(* IEC 61131-3 sources: pandora/pandora/aws-platform-main/aws-platform-main/configurations/base, 23 files *)

(* ---- Adaptio_IO.st ---- *)
USING Esab.Modes;

CONFIGURATION AdaptioIoMapping
    {::ifndef UNLINK_ADAPTIO_IO}
    VAR_GLOBAL
        // Adaptio
        {S7.Extern=ReadOnly}
        I_Adaptio AT %IB1000 : RawFromAdaptio;
        {S7.Extern=ReadOnly}
        Q_Adaptio AT %QB1000 : RawToAdaptio;
    END_VAR
    {::else}
    VAR_GLOBAL
        // Adaptio
        {S7.Extern=ReadWrite}
        I_Adaptio : RawFromAdaptio;
        {S7.Extern=ReadWrite}
        Q_Adaptio : RawToAdaptio;
    END_VAR
    {::endif}
END_CONFIGURATION

(* ---- B_IO.st ---- *)
USING Esab.Io;
USING Esab.WeldSystem.PowerSources;

CONFIGURATION BIoMapping
    {::ifndef UNLINK_B_IO}
    VAR_GLOBAL
        // -- B70 (Main I/O in B-cabinet) input/output starts at %X100

        // B71.1
        DI_B_System_CircuitBreaker_ServoDrives_OK AT %I100.0 : BOOL;
        DI_B_System_CircuitBreaker_ExternalConsumers_OK AT %I100.1 : BOOL;
        DI_B_System_EmergencyStop_OK AT %I100.2 : BOOL;
        DI_B_System_AirPressure_OK AT %I100.3 : BOOL;
        DI_B_RollerBed_External_Error AT %I100.4 : BOOL;
        /// Emergency stop reset button (B-cabinet)
        DI_B_PushButton_EmergencyStop_Reset AT %I100.5 : BOOL;
        // DI_SPARE AT %I100.6 : BOOL;
        // DI_SPARE AT %I100.7 : BOOL;
        DI_B_SpeedWheel_OneTurnSwitch AT %I101.0 : BOOL;
        DI_B_FluxSystem_Error AT %I101.1 : BOOL;
        DI_B_ClimateControl_Alarm AT %I101.2 : BOOL;
        // DI_SPARE AT %I101.3 : BOOL;
        // DI_SPARE AT %I101.4 : BOOL;
        // DI_SPARE AT %I101.5 : BOOL;
        // DI_SPARE AT %I101.6 : BOOL;
        // DI_SPARE AT %I101.7 : BOOL;

        // B71.2
        DI_B_PushButton_PusherRemote_WireFeed1_Down AT %I102.0 : BOOL;
        DI_B_PushButton_PusherRemote_WireFeed1_Up AT %I102.1 : BOOL;
        DI_B_PushButton_PusherRemote_WireFeed1_HighSpeed AT %I102.2 : BOOL;
        DI_B_PushButton_PusherRemote_WireFeed2_Down AT %I102.3 : BOOL;
        DI_B_PushButton_PusherRemote_WireFeed2_Up AT %I102.4 : BOOL;
        DI_B_PushButton_PusherRemote_WireFeed2_HighSpeed AT %I102.5 : BOOL;
        DI_B_PushButton_PusherRemote_WireFeed3_Down AT %I102.6 : BOOL;
        DI_B_PushButton_PusherRemote_WireFeed3_Up AT %I102.7 : BOOL;
        DI_B_PushButton_PusherRemote_WireFeed3_HighSpeed AT %I103.0 : BOOL;
        // DI_SPARE AT %I103.1 : BOOL;
        // DI_SPARE AT %I103.2 : BOOL;
        // DI_SPARE AT %I103.3 : BOOL;
        // DI_SPARE AT %I103.4 : BOOL;
        // DI_SPARE AT %I103.5 : BOOL;
        // DI_SPARE AT %I103.6 : BOOL;
        // DI_SPARE AT %I103.7 : BOOL;

        // B72.1
        DQ_B_PowerSource1_RemoteStart AT %Q100.0 : BOOL;
        DQ_B_PowerSource2_RemoteStart AT %Q100.1 : BOOL;
        DQ_B_PowerSource3_RemoteStart AT %Q100.2 : BOOL;
        DQ_B_System_RotatingWarningLight AT %Q100.3 : BOOL;
        DQ_B_FluxSystem_LowFluxWarningLight AT %Q100.4 : BOOL;
        /// This sets the reset signal to the safety relay in cabinet B.
        /// Do not use until safety investigation is complete.
        DQ_B_System_EmergencyStop_Reset AT %Q100.5 : BOOL;
        DQ_B_HighSpeed_Indicators AT %Q100.6 : BOOL;
        // DQ_SPARE AT Q100.7 : BOOL;
        // DQ_SPARE AT Q101.0 : BOOL;
        // DQ_SPARE AT Q101.1 : BOOL;
        // DQ_SPARE AT Q101.2 : BOOL;
        // DQ_SPARE AT Q101.3 : BOOL;
        // DQ_SPARE AT Q101.4 : BOOL;
        // DQ_SPARE AT Q101.5 : BOOL;
        // DQ_SPARE AT Q101.6 : BOOL;
        // DQ_SPARE AT Q101.7 : BOOL;

        // B73.1
        AI_B_EdgeSensor_Value AT %IW104 : INT;
        //AI_SPARE AT %IW106 : INT;
        //AI_SPARE AT %IW108 : INT;
        //AI_SPARE AT %IW110 : INT;

        // B74.1
        AI_B_FluxSystem_Temperature AT %IW112 : INT;
        //AI_SPARE AT %IW114 : INT;
        //AI_SPARE AT %IW116 : INT;
        //AI_SPARE AT %IW118 : INT;

        // B75.1
        AQ_B_RollerBed_SpeedReference AT %QW102 : INT;
        // AQ_SPARE AT %Q104 : INT;

        // B76.1
        DQ_B_RollerBed_Forward AT %Q106.0 : BOOL;
        DQ_B_RollerBed_Reverse AT %Q106.1 : BOOL;
        DQ_B_RollerBed_RemoteControl AT %Q106.2 : BOOL;
        // DQ_SPARE AT %Q106.3 : BOOL;

        // B77.1
        I_HighSpeedCounter AT %IB120 : RawHighSpeedCounterInputs;
        Q_HighSpeedCounter AT %QB107 : RawHighSpeedCounterOutputs;

        // B78.1
        DI_B_WireFeed1_PusherEncoder_A AT %I136.0 : BOOL;
        DI_B_WireFeed2_PusherEncoder_A AT %I136.1 : BOOL;
        DI_B_WireFeed3_PusherEncoder_A AT %I136.2 : BOOL;
        // DI_SPARE AT %I136.3 : BOOL;
        DI_B_WireFeed1_PusherEncoder_B AT %I136.4 : BOOL;
        DI_B_WireFeed2_PusherEncoder_B AT %I136.5 : BOOL;
        DI_B_WireFeed3_PusherEncoder_B AT %I136.6 : BOOL;
    END_VAR
    {::else}
    VAR_GLOBAL
        // -- B70 (Main I/O in B-cabinet) input/output starts at %X100

        // B71.1
        {S7.Extern=ReadWrite}
        DI_B_System_CircuitBreaker_ServoDrives_OK : BOOL;
        {S7.Extern=ReadWrite}
        DI_B_System_CircuitBreaker_ExternalConsumers_OK : BOOL;
        {S7.Extern=ReadWrite}
        DI_B_System_EmergencyStop_OK : BOOL;
        {S7.Extern=ReadWrite}
        DI_B_System_AirPressure_OK : BOOL;
        {S7.Extern=ReadWrite}
        DI_B_RollerBed_External_Error : BOOL;
        /// Emergency stop reset button (B-cabinet)
        {S7.Extern=ReadWrite}
        DI_B_PushButton_EmergencyStop_Reset : BOOL;
        // DI_SPARE AT %I100.6 : BOOL;
        // DI_SPARE AT %I100.7 : BOOL;
        {S7.Extern=ReadWrite}
        DI_B_SpeedWheel_OneTurnSwitch : BOOL;
        {S7.Extern=ReadWrite}
        DI_B_FluxSystem_Error : BOOL;
        {S7.Extern=ReadWrite}
        DI_B_ClimateControl_Alarm : BOOL;
        // DI_SPARE AT %I101.3 : BOOL;
        // DI_SPARE AT %I101.4 : BOOL;
        // DI_SPARE AT %I101.5 : BOOL;
        // DI_SPARE AT %I101.6 : BOOL;
        // DI_SPARE AT %I101.7 : BOOL;

        // B71.2
        {S7.Extern=ReadWrite}
        DI_B_PushButton_PusherRemote_WireFeed1_Down : BOOL;
        {S7.Extern=ReadWrite}
        DI_B_PushButton_PusherRemote_WireFeed1_Up : BOOL;
        {S7.Extern=ReadWrite}
        DI_B_PushButton_PusherRemote_WireFeed1_HighSpeed : BOOL;
        {S7.Extern=ReadWrite}
        DI_B_PushButton_PusherRemote_WireFeed2_Down : BOOL;
        {S7.Extern=ReadWrite}
        DI_B_PushButton_PusherRemote_WireFeed2_Up : BOOL;
        {S7.Extern=ReadWrite}
        DI_B_PushButton_PusherRemote_WireFeed2_HighSpeed : BOOL;
        {S7.Extern=ReadWrite}
        DI_B_PushButton_PusherRemote_WireFeed3_Down : BOOL;
        {S7.Extern=ReadWrite}
        DI_B_PushButton_PusherRemote_WireFeed3_Up : BOOL;
        {S7.Extern=ReadWrite}
        DI_B_PushButton_PusherRemote_WireFeed3_HighSpeed : BOOL;
        // DI_SPARE AT %I103.1 : BOOL;
        // DI_SPARE AT %I103.2 : BOOL;
        // DI_SPARE AT %I103.3 : BOOL;
        // DI_SPARE AT %I103.4 : BOOL;
        // DI_SPARE AT %I103.5 : BOOL;
        // DI_SPARE AT %I103.6 : BOOL;
        // DI_SPARE AT %I103.7 : BOOL;

        // B72.1
        {S7.Extern=ReadWrite}
        DQ_B_PowerSource1_RemoteStart : BOOL;
        {S7.Extern=ReadWrite}
        DQ_B_PowerSource2_RemoteStart : BOOL;
        {S7.Extern=ReadWrite}
        DQ_B_PowerSource3_RemoteStart : BOOL;
        {S7.Extern=ReadWrite}
        DQ_B_System_RotatingWarningLight : BOOL;
        {S7.Extern=ReadWrite}
        DQ_B_FluxSystem_LowFluxWarningLight : BOOL;
        /// This sets the reset signal to the safety relay in cabinet B.
        /// Do not use until safety investigation is complete.
        {S7.Extern=ReadWrite}
        DQ_B_System_EmergencyStop_Reset : BOOL;
        {S7.Extern=ReadWrite}
        DQ_B_HighSpeed_Indicators : BOOL;
        // DQ_SPARE AT Q100.7 : BOOL;
        // DQ_SPARE AT Q101.0 : BOOL;
        // DQ_SPARE AT Q101.1 : BOOL;
        // DQ_SPARE AT Q101.2 : BOOL;
        // DQ_SPARE AT Q101.3 : BOOL;
        // DQ_SPARE AT Q101.4 : BOOL;
        // DQ_SPARE AT Q101.5 : BOOL;
        // DQ_SPARE AT Q101.6 : BOOL;
        // DQ_SPARE AT Q101.7 : BOOL;

        // B73.1
        {S7.Extern=ReadWrite}
        AI_B_EdgeSensor_Value : INT;
        //AI_SPARE AT %IW106 : INT;
        //AI_SPARE AT %IW108 : INT;
        //AI_SPARE AT %IW110 : INT;

        // B74.1
        {S7.Extern=ReadWrite}
        AI_B_FluxSystem_Temperature : INT;
        //AI_SPARE AT %IW114 : INT;
        //AI_SPARE AT %IW116 : INT;
        //AI_SPARE AT %IW118 : INT;

        // B75.1
        {S7.Extern=ReadWrite}
        AQ_B_RollerBed_SpeedReference : INT;
        // AQ_SPARE AT %Q104 : INT;

        // B76.1
        {S7.Extern=ReadWrite}
        DQ_B_RollerBed_Forward : BOOL;
        {S7.Extern=ReadWrite}
        DQ_B_RollerBed_Reverse : BOOL;
        {S7.Extern=ReadWrite}
        DQ_B_RollerBed_RemoteControl : BOOL;
        // DQ_SPARE AT %Q106.3 : BOOL;

        // B77.1
        {S7.Extern=ReadWrite}
        I_HighSpeedCounter AT %MB100 : RawHighSpeedCounterInputs;
        {S7.Extern=ReadWrite}
        Q_HighSpeedCounter AT %MB150: RawHighSpeedCounterOutputs;

        // B78.1
        {S7.Extern=ReadWrite}
        DI_B_WireFeed1_PusherEncoder_A : BOOL;
        {S7.Extern=ReadWrite}
        DI_B_WireFeed2_PusherEncoder_A : BOOL;
        {S7.Extern=ReadWrite}
        DI_B_WireFeed3_PusherEncoder_A : BOOL;
        // DI_SPARE AT %I136.3 : BOOL;
        {S7.Extern=ReadWrite}
        DI_B_WireFeed1_PusherEncoder_B : BOOL;
        {S7.Extern=ReadWrite}
        DI_B_WireFeed2_PusherEncoder_B : BOOL;
        {S7.Extern=ReadWrite}
        DI_B_WireFeed3_PusherEncoder_B : BOOL;
    END_VAR
    {::endif}

END_CONFIGURATION

(* ---- C_IO.st ---- *)
CONFIGURATION CIoMapping
    {::ifndef UNLINK_C_IO}
    VAR_GLOBAL
        // -- C1 (Button box located at welding head) input/output starts at %X50
        // NOTE: The actual buttons are in the reverse order compared to I/O-addressing

        // C2
        /// Emergency stop reset button (C-cabinet)
        DI_C_PushButton_EmergencyStop_Reset AT %I59.0 : BOOL;
        /// Emergency stop reset button LED (C-cabinet)
        DQ_C_PushButton_EmergencyStop_Reset AT %Q59.0 : BOOL;

        // C3
        DI_C_PushButton_FluxSystem_Release AT %I58.0 : BOOL;
        DQ_C_PushButton_FluxSystem_Release AT %Q58.0 : BOOL;

        // C4
        DI_C_PushButton_HighSpeed AT %I57.0 : BOOL;
        DQ_C_PushButton_HighSpeed AT %Q57.0 : BOOL;

        // C5
        DI_C_PushButton_WireFeed1_Up AT %I56.0 : BOOL;
        DI_C_PushButton_WireFeed1_Down AT %I56.1 : BOOL;

        // C6
        DI_C_PushButton_WireFeed2_Up AT %I55.0 : BOOL;
        DI_C_PushButton_WireFeed2_Down AT %I55.1 : BOOL;

        // C7
        DI_C_PushButton_WireFeed3_Up AT %I54.0 : BOOL;
        DI_C_PushButton_WireFeed3_Down AT %I54.1 : BOOL;

        // C8 (Joystick) + C9 (Wired to the command module)
        DI_C_PushButton_TrackingOff AT %I50.0 : BOOL;
        DQ_C_PushButton_TrackingOff AT %Q50.0 : BOOL;
        DI_C_MotionJoystick_Up AT %I50.2 : BOOL;
        DI_C_MotionJoystick_Down AT %I50.3 : BOOL;
        DI_C_MotionJoystick_Triangle AT %I50.4 : BOOL;
        DI_C_MotionJoystick_Square AT %I50.5 : BOOL;

        // C10
        DI_C_PushButton_Tilt_Left AT %I53.0 : BOOL;
        DI_C_PushButton_Tilt_Right AT %I53.1 : BOOL;
    END_VAR
    {::else}
    VAR_GLOBAL
        // -- C1 (Button box located at welding head) input/output starts at %X50
        // NOTE: The actual buttons are in the reverse order compared to I/O-addressing

        // C2
        /// Emergency stop reset button (C-cabinet)
        {S7.Extern=ReadWrite}
        DI_C_PushButton_EmergencyStop_Reset : BOOL;
        /// Emergency stop reset button LED (C-cabinet)
        {S7.Extern=ReadWrite}
        DQ_C_PushButton_EmergencyStop_Reset : BOOL;

        // C3
        {S7.Extern=ReadWrite}
        DI_C_PushButton_FluxSystem_Release : BOOL;
        {S7.Extern=ReadWrite}
        DQ_C_PushButton_FluxSystem_Release : BOOL;

        // C4
        {S7.Extern=ReadWrite}
        DI_C_PushButton_HighSpeed : BOOL;
        {S7.Extern=ReadWrite}
        DQ_C_PushButton_HighSpeed : BOOL;

        // C5
        {S7.Extern=ReadWrite}
        DI_C_PushButton_WireFeed1_Up : BOOL;
        {S7.Extern=ReadWrite}
        DI_C_PushButton_WireFeed1_Down : BOOL;

        // C6
        {S7.Extern=ReadWrite}
        DI_C_PushButton_WireFeed2_Up : BOOL;
        {S7.Extern=ReadWrite}
        DI_C_PushButton_WireFeed2_Down : BOOL;

        // C7
        {S7.Extern=ReadWrite}
        DI_C_PushButton_WireFeed3_Up : BOOL;
        {S7.Extern=ReadWrite}
        DI_C_PushButton_WireFeed3_Down : BOOL;

        // C8 (Joystick) + C9 (Wired to the command module)
        {S7.Extern=ReadWrite}
        DI_C_PushButton_TrackingOff : BOOL;
        {S7.Extern=ReadWrite}
        DQ_C_PushButton_TrackingOff : BOOL;
        {S7.Extern=ReadWrite}
        DI_C_MotionJoystick_Up : BOOL;
        {S7.Extern=ReadWrite}
        DI_C_MotionJoystick_Down : BOOL;
        {S7.Extern=ReadWrite}
        DI_C_MotionJoystick_Triangle : BOOL;
        {S7.Extern=ReadWrite}
        DI_C_MotionJoystick_Square : BOOL;

        // C10
        {S7.Extern=ReadWrite}
        DI_C_PushButton_Tilt_Left : BOOL;
        {S7.Extern=ReadWrite}
        DI_C_PushButton_Tilt_Right : BOOL;
    END_VAR
    {::endif}
END_CONFIGURATION

(* ---- GlobalState.st ---- *)
USING Esab.WeldSystem.Flux;
USING Esab.Utils.Alarming;
USING Esab.Utils.Assets;
USING Esab.Modes;

USING Siemens.Simatic.S71500.Tasks;
USING Siemens.Simatic.S71500.Alarming;

CONFIGURATION GlobalStateConfiguration

    // Constants
    VAR_GLOBAL CONSTANT
    END_VAR

    // Objects
    VAR_GLOBAL
        {S7.Extern=Read}
        GlobalState : Esab.GlobalState;
    END_VAR

    // Alarms
    VAR_GLOBAL
        GlobalStateSetupAlarmWrapper : AlarmWrapper;
        {S7.Alarm = NoAck, "Global state: Setup error."}
        GlobalStateSetupAlarm : ProgramAlarm;
    END_VAR

    // Interface
    VAR_GLOBAL
    END_VAR
END_CONFIGURATION

FUNCTION InitializeGlobalState
    VAR_INPUT
        assetsManager : IAssetsManager;
    END_VAR

    VAR_EXTERNAL
        GlobalState : Esab.GlobalState;

        GlobalStateSetupAlarmWrapper : AlarmWrapper;
        GlobalStateSetupAlarm : ProgramAlarm;
    END_VAR

    GlobalStateSetupAlarmWrapper.Setup(REF(GlobalStateSetupAlarm));

    GlobalState.Setup(assetsManager, GlobalStateSetupAlarmWrapper);

    GlobalState.SetIdentifier(Esab.AssetIdentifier#GlobalState);
    assetsManager.RegisterAsset(REF(GlobalState));

    // By default we set the GlobalState mode to be Adaptio
    GlobalState.SetMode(Esab.AwsPlatformMode#Adaptio);
END_FUNCTION

(* ---- H_IO.st ---- *)
CONFIGURATION HIoMapping
    {::ifndef UNLINK_H_IO}
    VAR_GLOBAL
        // -- H1 (Weld head I/O) input/output starts at %X60

        // H2.1
        DI_H_SlideCrossHorizontal_LimitSwitch_Triangle AT %I60.0 : BOOL;
        DI_H_SlideCrossHorizontal_LimitSwitch_Square AT %I60.1 : BOOL;
        DI_H_SlideCrossVertical_LimitSwitch_Up AT %I60.2 : BOOL;
        DI_H_SlideCrossVertical_LimitSwitch_Down AT %I60.3 : BOOL;
        DI_H_Tilt_LimitSwitch_Left AT %I60.4 : BOOL;
        DI_H_Tilt_LimitSwitch_Right AT %I60.5 : BOOL;
        // DI_SPARE AT %I60.6 : BOOL;
        // DI_SPARE AT %I60.7 : BOOL;

        // H3.1
        AI_H_Pyrometer_Value AT %IW61 : INT;
        AI_H_HeightSensor_Value AT %IW63 : INT;
        // AI_SPARE AT %IW65 : INT;
        // AI_SPARE AT %IW67 : INT;

        // H4.1
        DQ_H_LaserPointer_Enable AT %Q69.0 : BOOL;
        DQ_H_System_Water_WarningLight AT %Q69.1 : BOOL;
        // DQ_SPARE AT %!69.2 : BOOL;
        // DQ_SPARE AT %!69.3 : BOOL;
        // DQ_SPARE AT %!69.4 : BOOL;
        // DQ_SPARE AT %!69.5 : BOOL;
        DQ_H_Scanner_LaserLine_Enable AT %Q69.6 : BOOL;
        DQ_H_Scanner_Camera_Enable AT %Q69.7 : BOOL;

        // H4.2
        DQ_H_FluxSystem_Recover AT %Q70.0 : BOOL;
        DQ_H_FluxSystem_Release AT %Q70.1 : BOOL;
        DQ_H_Scanner_AirFlow_Enable AT %Q70.2 : BOOL;
        DQ_H_FluxSystem_NozzleRotation AT %Q70.3 : BOOL;
        // DQ_SPARE AT %Q70.4 : BOOL;
        // DQ_SPARE AT %Q70.5 : BOOL;
        // DQ_SPARE AT %Q70.6 : BOOL;
        // DQ_SPARE AT %Q70.7 : BOOL;

        // H5.1
        DQ_H_Camera_Lamp1_Enable AT %Q71.0 : BOOL;
        DQ_H_Camera_Lamp2_Enable AT %Q71.1 : BOOL;
        DQ_H_FloodLight1_Enable AT %Q71.2 : BOOL;
        DQ_H_FloodLight2_Enable AT %Q71.3 : BOOL;
    END_VAR
    {::else}
    VAR_GLOBAL
        // -- H1 (Weld head I/O) input/output starts at %X60

        // H2.1
        {S7.Extern=ReadWrite}
        DI_H_SlideCrossHorizontal_LimitSwitch_Triangle : BOOL;
        {S7.Extern=ReadWrite}
        DI_H_SlideCrossHorizontal_LimitSwitch_Square : BOOL;
        {S7.Extern=ReadWrite}
        DI_H_SlideCrossVertical_LimitSwitch_Up : BOOL;
        {S7.Extern=ReadWrite}
        DI_H_SlideCrossVertical_LimitSwitch_Down : BOOL;
        {S7.Extern=ReadWrite}
        DI_H_Tilt_LimitSwitch_Left : BOOL;
        {S7.Extern=ReadWrite}
        DI_H_Tilt_LimitSwitch_Right : BOOL;
        // DI_SPARE AT %I60.6 : BOOL;
        // DI_SPARE AT %I60.7 : BOOL;

        // H3.1
        {S7.Extern=ReadWrite}
        AI_H_Pyrometer_Value : INT;
        {S7.Extern=ReadWrite}
        AI_H_HeightSensor_Value : INT;
        // AI_SPARE AT %IW65 : INT;
        // AI_SPARE AT %IW67 : INT;

        // H4.1
        {S7.Extern=ReadWrite}
        DQ_H_LaserPointer_Enable : BOOL;
        {S7.Extern=ReadWrite}
        DQ_H_System_Water_WarningLight : BOOL;
        // DQ_SPARE AT %!69.2 : BOOL;
        // DQ_SPARE AT %!69.3 : BOOL;
        // DQ_SPARE AT %!69.4 : BOOL;
        // DQ_SPARE AT %!69.5 : BOOL;
        {S7.Extern=ReadWrite}
        DQ_H_Scanner_LaserLine_Enable : BOOL;
        {S7.Extern=ReadWrite}
        DQ_H_Scanner_Camera_Enable : BOOL;

        // H4.2
        {S7.Extern=ReadWrite}
        DQ_H_FluxSystem_Recover : BOOL;
        {S7.Extern=ReadWrite}
        DQ_H_FluxSystem_Release : BOOL;
        {S7.Extern=ReadWrite}
        DQ_H_Scanner_AirFlow_Enable : BOOL;
        {S7.Extern=ReadWrite}
        DQ_H_FluxSystem_NozzleRotation : BOOL;
        // DQ_SPARE AT %Q70.4 : BOOL;
        // DQ_SPARE AT %Q70.5 : BOOL;
        // DQ_SPARE AT %Q70.6 : BOOL;
        // DQ_SPARE AT %Q70.7 : BOOL;

        // H5.1
        {S7.Extern=ReadWrite}
        DQ_H_Camera_Lamp1_Enable : BOOL;
        {S7.Extern=ReadWrite}
        DQ_H_Camera_Lamp2_Enable : BOOL;
        {S7.Extern=ReadWrite}
        DQ_H_FloodLight1_Enable : BOOL;
        {S7.Extern=ReadWrite}
        DQ_H_FloodLight2_Enable : BOOL;
    END_VAR
    {::endif}
END_CONFIGURATION

(* ---- P_IO.st ---- *)
CONFIGURATION IoMapping
    {::ifndef UNLINK_P_IO}
    VAR_GLOBAL
        // -- P1 (Button box below the main HMI screen) input/output starts at %X30
        // NOTE: The actual buttons are in the reverse order compared to I/O-addressing

        // P2 (Emergency stop reset)
        DI_P_PushButton_EmergencyStop_Reset AT %I42.0 : BOOL;
        DQ_P_PushButton_EmergencyStop_Reset AT %Q42.0 : BOOL;

        // P3 (Flux release/down)
        DI_P_PushButton_FluxSystem_Release AT %I41.0 : BOOL;
        DQ_P_PushButton_FluxSystem_Release AT %Q41.0 : BOOL;

        // P4 (Flux recover/suction)
        DI_P_PushButton_FluxSystem_Recover AT %I40.0 : BOOL;
        DQ_P_PushButton_FluxSystem_Recover AT %Q40.0 : BOOL;

        // P5 (High speed selection)
        DI_P_PushButton_HighSpeed AT %I39.0 : BOOL;
        DQ_P_PushButton_HighSpeed AT %Q39.0 : BOOL;

        // P6 (Wire feed 1 + 3)
        /// NOTE: This also controls WF 3 Up through mode select
        DI_P_PushButton_WireFeed1_Up AT %I38.0 : BOOL;
        /// NOTE: This also controls WF 3 Down through mode select
        DI_P_PushButton_WireFeed1_Down AT %I38.1 : BOOL;

        // P7
        DI_P_PushButton_WireFeed2_Up AT %I37.0 : BOOL;
        DI_P_PushButton_WireFeed2_Down AT %I37.1 : BOOL;

        // P8 (Joystick) + P9 (Axis selection)
        DI_P_MotionJoystick_AxisSelection AT %I30.0 : BOOL;
        DQ_P_MotionJoystick_AxisSelection AT %Q30.0 : BOOL;
        DI_P_MotionJoystick_Up AT %I30.2 : BOOL;
        DI_P_MotionJoystick_Down AT %I30.3 : BOOL;
        DI_P_MotionJoystick_Triangle AT %I30.4 : BOOL;
        DI_P_MotionJoystick_Square AT %I30.5 : BOOL;

        // P10 (Axis selection triangle/square)
        DI_P_PushButton_AxisJog_AxisSelection AT %I36.0 : BOOL;
        DQ_P_PushButton_AxisJog_AxisSelection AT %Q36.0 : BOOL;

        // P11 (Axis triangle/square)
        DI_P_PushButton_AxisJog_Triangle AT %I35.0 : BOOL;
        DI_P_PushButton_AxisJog_Square AT %I35.1 : BOOL;

        // P12 (Start)
        DI_P_PushButton_Start AT %I34.0 : BOOL;
        DQ_P_PushButton_Start AT %Q34.0 : BOOL;

        // P13 (Stop)
        DI_P_PushButton_Stop AT %I33.0 : BOOL;
        DQ_P_PushButton_Stop AT %Q33.0 : BOOL;
    END_VAR
    {::else}
    VAR_GLOBAL
        // -- P1 (Button box below the main HMI screen) input/output starts at %X30
        // NOTE: The actual buttons are in the reverse order compared to I/O-addressing

        // P2 (Emergency stop reset)
        {S7.Extern=ReadWrite}
        DI_P_PushButton_EmergencyStop_Reset : BOOL;
        {S7.Extern=ReadWrite}
        DQ_P_PushButton_EmergencyStop_Reset : BOOL;

        // P3 (Flux release/down)
        {S7.Extern=ReadWrite}
        DI_P_PushButton_FluxSystem_Release : BOOL;
        {S7.Extern=ReadWrite}
        DQ_P_PushButton_FluxSystem_Release : BOOL;

        // P4 (Flux recover/suction)
        {S7.Extern=ReadWrite}
        DI_P_PushButton_FluxSystem_Recover : BOOL;
        {S7.Extern=ReadWrite}
        DQ_P_PushButton_FluxSystem_Recover : BOOL;

        // P5 (High speed selection)
        {S7.Extern=ReadWrite}
        DI_P_PushButton_HighSpeed : BOOL;
        {S7.Extern=ReadWrite}
        DQ_P_PushButton_HighSpeed : BOOL;

        // P6 (Wire feed 1 + 3)
        /// NOTE: This also controls WF 3 Up through mode select
        {S7.Extern=ReadWrite}
        DI_P_PushButton_WireFeed1_Up : BOOL;
        /// NOTE: This also controls WF 3 Down through mode select
        {S7.Extern=ReadWrite}
        DI_P_PushButton_WireFeed1_Down : BOOL;

        // P7
        {S7.Extern=ReadWrite}
        DI_P_PushButton_WireFeed2_Up : BOOL;
        {S7.Extern=ReadWrite}
        DI_P_PushButton_WireFeed2_Down : BOOL;

        // P8 (Joystick) + P9 (Axis selection)
        {S7.Extern=ReadWrite}
        DI_P_MotionJoystick_AxisSelection : BOOL;
        {S7.Extern=ReadWrite}
        DQ_P_MotionJoystick_AxisSelection : BOOL;
        {S7.Extern=ReadWrite}
        DI_P_MotionJoystick_Up : BOOL;
        {S7.Extern=ReadWrite}
        DI_P_MotionJoystick_Down : BOOL;
        {S7.Extern=ReadWrite}
        DI_P_MotionJoystick_Triangle : BOOL;
        {S7.Extern=ReadWrite}
        DI_P_MotionJoystick_Square : BOOL;

        // P10 (Axis selection triangle/square)
        {S7.Extern=ReadWrite}
        DI_P_PushButton_AxisJog_AxisSelection : BOOL;
        {S7.Extern=ReadWrite}
        DQ_P_PushButton_AxisJog_AxisSelection : BOOL;

        // P11 (Axis triangle/square)
        {S7.Extern=ReadWrite}
        DI_P_PushButton_AxisJog_Triangle : BOOL;
        {S7.Extern=ReadWrite}
        DI_P_PushButton_AxisJog_Square : BOOL;

        // P12 (Start)
        {S7.Extern=ReadWrite}
        DI_P_PushButton_Start : BOOL;
        {S7.Extern=ReadWrite}
        DQ_P_PushButton_Start : BOOL;

        // P13 (Stop)
        {S7.Extern=ReadWrite}
        DI_P_PushButton_Stop : BOOL;
        {S7.Extern=ReadWrite}
        DQ_P_PushButton_Stop : BOOL;
    END_VAR
    {::endif}
END_CONFIGURATION

(* ---- PowerSources_IO.st ---- *)
USING Esab.WeldSystem.PowerSources;

CONFIGURATION PowerSourcesIoMapping
    {::ifndef UNLINK_POWERSOURCES_IO}
    VAR_GLOBAL
        // Power sources
        I_Pab1 AT %IB500 : RawPabToController;
        Q_Pab1 AT %QB500 : RawControllerToPab;
        I_Pab2 AT %IB600 : RawPabToController;
        Q_Pab2 AT %QB600 : RawControllerToPab;
    END_VAR
    {::else}
    VAR_GLOBAL
        // Power sources
        {S7.Extern=ReadWrite}
        I_Pab1 : RawPabToController;
        {S7.Extern=ReadWrite}
        Q_Pab1 : RawControllerToPab;
        {S7.Extern=ReadWrite}
        I_Pab2 : RawPabToController;
        {S7.Extern=ReadWrite}
        Q_Pab2 : RawControllerToPab;
    END_VAR
    {::endif}
END_CONFIGURATION

(* ---- SlideCrossAxis.st ---- *)
USING Esab.Motion;
USING Esab.Utils.Assets;

CONFIGURATION SlideCrossConfiguration
    // Constants
    VAR_GLOBAL CONSTANT
        HORIZONTAL_SLIDE_AXIS_DB : Siemens.Simatic.S71500.MotionControl.Native.DB_ANY := UINT#1;
        VERTICAL_SLIDE_AXIS_DB : Siemens.Simatic.S71500.MotionControl.Native.DB_ANY := UINT#2;
    END_VAR

    // Objects
    VAR_GLOBAL
        Technology : TechnologyObjects;
        HorizontalSlideAxis : ToPosAxis;
        HorizontalSlideAxisRuntimeParameters : AxisRuntimeParameters;
        VerticalSlideAxis : ToPosAxis;
        VerticalSlideAxisRuntimeParameters : AxisRuntimeParameters;
    END_VAR

    // Alarms
    VAR_GLOBAL
    END_VAR

    // Interface
    VAR_GLOBAL
    END_VAR
END_CONFIGURATION

FUNCTION InitializeSlideCrossAxis
    VAR_INPUT
        assetsManager : IAssetsManager;
    END_VAR

    VAR_EXTERNAL CONSTANT
        HORIZONTAL_SLIDE_AXIS_DB : Siemens.Simatic.S71500.MotionControl.Native.DB_ANY;
        VERTICAL_SLIDE_AXIS_DB : Siemens.Simatic.S71500.MotionControl.Native.DB_ANY;
    END_VAR

    VAR_EXTERNAL
        Technology : TechnologyObjects;
        HorizontalSlideAxis : ToPosAxis;
        HorizontalSlideAxisRuntimeParameters : AxisRuntimeParameters;
        VerticalSlideAxis : ToPosAxis;
        VerticalSlideAxisRuntimeParameters : AxisRuntimeParameters;
    END_VAR

    Technology.Setup(HORIZONTAL_SLIDE_AXIS_DB, VERTICAL_SLIDE_AXIS_DB);

    IF Technology.IsAttached() THEN
        HorizontalSlideAxis.Setup(Technology.GetHorizontalSlideAxis(), REF(HorizontalSlideAxisRuntimeParameters));
        VerticalSlideAxis.Setup(Technology.GetVerticalSlideAxis(), REF(VerticalSlideAxisRuntimeParameters));

        HorizontalSlideAxis.SetIdentifier(Esab.AssetIdentifier#HorizontalSlideAxis);
        VerticalSlideAxis.SetIdentifier(Esab.AssetIdentifier#VerticalSlideAxis);
        assetsManager.RegisterAsset(REF(HorizontalSlideAxis));
        assetsManager.RegisterAsset(REF(VerticalSlideAxis));
    END_IF;
END_FUNCTION

(* ---- Ups1600_IO.st ---- *)
USING Esab.Utils.Power;

CONFIGURATION Ups1600IoMapping

    {::ifndef UNLINK_UPS_IO}
    VAR_GLOBAL
        {S7.Extern=ReadOnly}
        I_Ups AT %IB0 : RawFromUps1600;
    END_VAR
    {::else}
    VAR_GLOBAL
        {S7.Extern=ReadWrite}
        I_Ups : RawFromUps1600;
    END_VAR
    {::endif}

END_CONFIGURATION

(* ---- WeldHeadManipulator.st ---- *)
USING Esab.Utils.Alarming;
USING Esab.Utils.Assets;
USING Esab.Motion;

USING Siemens.Simatic.S71500.Tasks;
USING Siemens.Simatic.S71500.Alarming;

CONFIGURATION WeldHeadManipulatorConfiguration

    // Constants
    VAR_GLOBAL CONSTANT
    END_VAR

    // Objects
    VAR_GLOBAL
        {S7.Extern=Read}
        WeldHeadManipulator : WeldHeadManipulator;
    END_VAR

    // Alarms
    VAR_GLOBAL
        WeldHeadManipulatorSetupAlarmWrapper : AlarmWrapper;
        {S7.Alarm = NoAck, "Global state: Setup error."}
        WeldHeadManipulatorSetupAlarm : ProgramAlarm;
    END_VAR

    // Interface
    VAR_GLOBAL
    END_VAR

    VAR_GLOBAL RETAIN
        WeldHeadManipulatorRuntimeParameters : WeldHeadManipulatorRuntimeParameters;
        WeldHeadManipulatorHardwareConfiguration : WeldHeadManipulatorHardwareConfiguration;
    END_VAR
END_CONFIGURATION

FUNCTION InitializeWeldHeadManipulator
    VAR_INPUT
        assetsManager : IAssetsManager;
    END_VAR

    VAR_EXTERNAL
        WeldHeadManipulator : WeldHeadManipulator;
        WeldHeadManipulatorRuntimeParameters : WeldHeadManipulatorRuntimeParameters;
        WeldHeadManipulatorHardwareConfiguration : WeldHeadManipulatorHardwareConfiguration;

        WeldHeadManipulatorSetupAlarmWrapper : AlarmWrapper;
        WeldHeadManipulatorSetupAlarm : ProgramAlarm;
    END_VAR

    WeldHeadManipulatorSetupAlarmWrapper.Setup(REF(WeldHeadManipulatorSetupAlarm));

    WeldHeadManipulator.Setup(REF(WeldHeadManipulatorRuntimeParameters),
                              REF(WeldHeadManipulatorHardwareConfiguration),
                              assetsManager,
                              WeldHeadManipulatorSetupAlarmWrapper);

    WeldHeadManipulator.SetIdentifier(Esab.AssetIdentifier#WeldHeadManipulator);
    assetsManager.RegisterAsset(REF(WeldHeadManipulator));
END_FUNCTION

(* ---- WeldSystemOrchestrator.st ---- *)
USING Esab.Utils.Alarming;
USING Esab.Utils.Assets;
USING Esab.WeldSystem;

USING Siemens.Simatic.S71500.Alarming;

CONFIGURATION WeldSystemOrchestratorConfiguration

    // Constants
    VAR_GLOBAL CONSTANT
    END_VAR

    // Objects
    VAR_GLOBAL
        WeldSystemOrchestrator : WeldSystemOrchestrator;
    END_VAR

    // Alarms
    VAR_GLOBAL
        WeldSystemOrchestratorSetupAlarmWrapper : AlarmWrapper;
        {S7.Alarm = NoAck, "Weld system: Setup error."}
        WeldSystemOrchestratorSetupAlarm : ProgramAlarm;
    END_VAR

    // Interface
    VAR_GLOBAL
    END_VAR

    VAR_GLOBAL RETAIN
        WeldSystemOrchestratorRuntimeParameters : WeldSystemOrchestratorRuntimeParameters;
        WeldSystemOrchestratorHardwareConfiguration : WeldSystemOrchestratorHardwareConfiguration;
    END_VAR
END_CONFIGURATION

FUNCTION InitializeMultiWeldSystem
    VAR_INPUT
        assetsManager : IAssetsManager;
    END_VAR

    VAR_EXTERNAL
        WeldSystemOrchestrator : WeldSystemOrchestrator;
        WeldSystemOrchestratorRuntimeParameters : WeldSystemOrchestratorRuntimeParameters;
        WeldSystemOrchestratorHardwareConfiguration : WeldSystemOrchestratorHardwareConfiguration;
        WeldSystemOrchestratorSetupAlarmWrapper : AlarmWrapper;
        WeldSystemOrchestratorSetupAlarm : ProgramAlarm;
    END_VAR

    WeldSystemOrchestratorSetupAlarmWrapper.Setup(REF(WeldSystemOrchestratorSetupAlarm));

    WeldSystemOrchestrator.Setup(REF(WeldSystemOrchestratorRuntimeParameters),
                                 REF(WeldSystemOrchestratorHardwareConfiguration),
                                 assetsManager,
                                 WeldSystemOrchestratorSetupAlarmWrapper);

    WeldSystemOrchestrator.SetIdentifier(Esab.AssetIdentifier#WeldSystemOrchestrator);
    assetsManager.RegisterAsset(REF(WeldSystemOrchestrator));
END_FUNCTION

(* ---- Adaptio.st ---- *)
USING Esab.Modes;
USING Esab.Utils.Alarming;
USING Esab.Utils.Assets;
USING Esab.Utils.Heartbeat;
USING Esab.Utils.Timer;

USING Siemens.Simatic.S71500.Tasks;
USING Siemens.Simatic.S71500.Alarming;

CONFIGURATION AdaptioSystemConfiguration

    TASK AdaptioIoTask : ProgramCycle;

    PROGRAM AdaptioIoReadWrite WITH AdaptioIoTask: AdaptioIoReadWrite;

    // Constants
    VAR_GLOBAL CONSTANT
    END_VAR

    // Objects
    VAR_GLOBAL
        {S7.Extern=Read}
        Adaptio : Adaptio;
        AdaptioRuntimeParameters : AdaptioRuntimeParameters;
        AdaptioWeldSequence : AdaptioWeldSequence;
        AdaptioWeldSequenceStateTimer : ITimer;
        AdaptioHeartbeat : IncrementingHeartbeat;
        AdaptioRequestTimer : OnDelay;
        AdaptioJoystickClickTimer : OnDelay;
        AdaptioWeldingStateTimer : OnDelay;
        AdaptioHeartbeatTimer : OnDelay;
    END_VAR

    // Alarms
    VAR_GLOBAL
        AdaptioHeartbeatAlarmWrapper : AlarmWrapper;
        {S7.Alarm = NoAck, "Adaptio: Heartbeat missing."}
        AdaptioHeartbeatAlarm : ProgramAlarm;

        AdaptioSetupAlarmWrapper : AlarmWrapper;
        {S7.Alarm = NoAck, "Adaptio: Setup error."}
        AdaptioSetupAlarm : ProgramAlarm;
    END_VAR

    // Interface
    VAR_GLOBAL
        {S7.Extern=ReadWrite}
        AdaptioIo : AdaptioIo;
    END_VAR
END_CONFIGURATION

FUNCTION InitializeAdaptio
    VAR_INPUT
        assetsManager : IAssetsManager;
    END_VAR

    VAR_EXTERNAL
        AdaptioIo : AdaptioIo;

        Adaptio : Adaptio;
        AdaptioRuntimeParameters : AdaptioRuntimeParameters;
        AdaptioWeldSequence : AdaptioWeldSequence;
        AdaptioWeldSequenceStateTimer : ITimer;
        AdaptioHeartbeat : IncrementingHeartbeat;
        AdaptioRequestTimer : OnDelay;
        AdaptioJoystickClickTimer : OnDelay;
        AdaptioWeldingStateTimer : OnDelay;
        AdaptioHeartbeatTimer : OnDelay;

        AdaptioHeartbeatAlarmWrapper : AlarmWrapper;
        AdaptioHeartbeatAlarm : ProgramAlarm;

        AdaptioSetupAlarmWrapper : AlarmWrapper;
        AdaptioSetupAlarm : ProgramAlarm;
    END_VAR

    AdaptioWeldSequence.Setup(AdaptioWeldSequenceStateTimer); // Weld axis and orchestrator is set inside the Adaptio manager
    AdaptioHeartbeatAlarmWrapper.Setup(REF(AdaptioHeartbeatAlarm));
    AdaptioSetupAlarmWrapper.Setup(REF(AdaptioSetupAlarm));

    AdaptioHeartbeat.Setup(AdaptioIo.FromAdaptio.SystemControl.Heartbeat,
                           AdaptioIo.ToAdaptio.SystemControl.Heartbeat,
                           AdaptioHeartbeatTimer,
                           AdaptioHeartbeatAlarmWrapper);

    Adaptio.Setup(REF(AdaptioIo),
                  REF(AdaptioRuntimeParameters),
                  assetsManager,
                  AdaptioWeldSequence,
                  AdaptioHeartbeat,
                  AdaptioRequestTimer,
                  AdaptioJoystickClickTimer,
                  AdaptioSetupAlarmWrapper);
END_FUNCTION

PROGRAM AdaptioIoReadWrite
    VAR_EXTERNAL
        AdaptioIo : AdaptioIo;
        I_Adaptio : RawFromAdaptio;
        Q_Adaptio : RawToAdaptio;
    END_VAR

    AdaptioIo.FromAdaptio.SystemControl.Heartbeat.Read(I_Adaptio.SystemControl.Heartbeat);

    AdaptioIo.FromAdaptio.WeldControl.Start.Read(I_Adaptio.WeldControl.Start);
    AdaptioIo.FromAdaptio.WeldControl.Stop.Read(I_Adaptio.WeldControl.Stop);
    AdaptioIo.FromAdaptio.WeldControl.QuickStop.Read(I_Adaptio.WeldControl.QuickStop);

    AdaptioIo.FromAdaptio.PowerSource1.Enable.Read(I_Adaptio.PowerSource1.Enable);
    AdaptioIo.FromAdaptio.PowerSource1.ActiveAreaSelect.Read(I_Adaptio.PowerSource1.ActiveAreaSelect);
    AdaptioIo.FromAdaptio.PowerSource1.SwitchAreas.Read(I_Adaptio.PowerSource1.SwitchAreas);
    AdaptioIo.FromAdaptio.PowerSource1.Voltage.Read(I_Adaptio.PowerSource1.Voltage);
    AdaptioIo.FromAdaptio.PowerSource1.Current.Read(I_Adaptio.PowerSource1.Current);
    AdaptioIo.FromAdaptio.PowerSource1.WireSpeed.Read(I_Adaptio.PowerSource1.WireSpeed);
    AdaptioIo.FromAdaptio.PowerSource1.RegulationType.Read(I_Adaptio.PowerSource1.RegulationType);
    AdaptioIo.FromAdaptio.PowerSource1.WeldMethod.Read(I_Adaptio.PowerSource1.WeldMethod);
    AdaptioIo.FromAdaptio.PowerSource1.AcFrequency.Read(I_Adaptio.PowerSource1.AcFrequency);
    AdaptioIo.FromAdaptio.PowerSource1.AcBalance.Read(I_Adaptio.PowerSource1.AcBalance);
    AdaptioIo.FromAdaptio.PowerSource1.AcOffset.Read(I_Adaptio.PowerSource1.AcOffset);
    AdaptioIo.FromAdaptio.PowerSource1.AcPhaseShift.Read(I_Adaptio.PowerSource1.AcPhaseShift);
    AdaptioIo.FromAdaptio.PowerSource1.StartAdjust.Read(I_Adaptio.PowerSource1.StartAdjust);
    AdaptioIo.FromAdaptio.PowerSource1.RegulationDynamics.Read(I_Adaptio.PowerSource1.RegulationDynamics);
    AdaptioIo.FromAdaptio.PowerSource1.RegulationInductance.Read(I_Adaptio.PowerSource1.RegulationInductance);
    AdaptioIo.FromAdaptio.PowerSource1.IceWireSpeed.Read(I_Adaptio.PowerSource1.IceWireSpeed);

    AdaptioIo.FromAdaptio.PowerSource2.Enable.Read(I_Adaptio.PowerSource2.Enable);
    AdaptioIo.FromAdaptio.PowerSource2.ActiveAreaSelect.Read(I_Adaptio.PowerSource2.ActiveAreaSelect);
    AdaptioIo.FromAdaptio.PowerSource2.SwitchAreas.Read(I_Adaptio.PowerSource2.SwitchAreas);
    AdaptioIo.FromAdaptio.PowerSource2.Voltage.Read(I_Adaptio.PowerSource2.Voltage);
    AdaptioIo.FromAdaptio.PowerSource2.Current.Read(I_Adaptio.PowerSource2.Current);
    AdaptioIo.FromAdaptio.PowerSource2.WireSpeed.Read(I_Adaptio.PowerSource2.WireSpeed);
    AdaptioIo.FromAdaptio.PowerSource2.RegulationType.Read(I_Adaptio.PowerSource2.RegulationType);
    AdaptioIo.FromAdaptio.PowerSource2.WeldMethod.Read(I_Adaptio.PowerSource2.WeldMethod);
    AdaptioIo.FromAdaptio.PowerSource2.AcFrequency.Read(I_Adaptio.PowerSource2.AcFrequency);
    AdaptioIo.FromAdaptio.PowerSource2.AcBalance.Read(I_Adaptio.PowerSource2.AcBalance);
    AdaptioIo.FromAdaptio.PowerSource2.AcOffset.Read(I_Adaptio.PowerSource2.AcOffset);
    AdaptioIo.FromAdaptio.PowerSource2.AcPhaseShift.Read(I_Adaptio.PowerSource2.AcPhaseShift);
    AdaptioIo.FromAdaptio.PowerSource2.StartAdjust.Read(I_Adaptio.PowerSource2.StartAdjust);
    AdaptioIo.FromAdaptio.PowerSource2.RegulationDynamics.Read(I_Adaptio.PowerSource2.RegulationDynamics);
    AdaptioIo.FromAdaptio.PowerSource2.RegulationInductance.Read(I_Adaptio.PowerSource2.RegulationInductance);
    AdaptioIo.FromAdaptio.PowerSource2.IceWireSpeed.Read(I_Adaptio.PowerSource2.IceWireSpeed);

    AdaptioIo.FromAdaptio.WeldAxis.EnableMotion.Read(I_Adaptio.WeldAxis.EnableMotion);
    AdaptioIo.FromAdaptio.WeldAxis.Reset.Read(I_Adaptio.WeldAxis.Reset);
    AdaptioIo.FromAdaptio.WeldAxis.InvalidateReference.Read(I_Adaptio.WeldAxis.InvalidateReference);
    AdaptioIo.FromAdaptio.WeldAxis.ResetLinearObjectDistance.Read(I_Adaptio.WeldAxis.ResetLinearObjectDistance);
    AdaptioIo.FromAdaptio.WeldAxis.MovementType.Read(I_Adaptio.WeldAxis.MovementType);
    AdaptioIo.FromAdaptio.WeldAxis.MovementMode.Read(I_Adaptio.WeldAxis.MovementMode);
    AdaptioIo.FromAdaptio.WeldAxis.Radius.Read(I_Adaptio.WeldAxis.Radius);
    AdaptioIo.FromAdaptio.WeldAxis.Position.Read(I_Adaptio.WeldAxis.Position);
    AdaptioIo.FromAdaptio.WeldAxis.Velocity.Read(I_Adaptio.WeldAxis.Velocity);

    AdaptioIo.FromAdaptio.WeldHeadManipulator.EnableMotion.Read(I_Adaptio.WeldHeadManipulator.EnableMotion);
    AdaptioIo.FromAdaptio.WeldHeadManipulator.Interpolate.Read(I_Adaptio.WeldHeadManipulator.Interpolate);
    AdaptioIo.FromAdaptio.WeldHeadManipulator.XPosition.Read(I_Adaptio.WeldHeadManipulator.XPosition);
    AdaptioIo.FromAdaptio.WeldHeadManipulator.YPosition.Read(I_Adaptio.WeldHeadManipulator.YPosition);
    AdaptioIo.FromAdaptio.WeldHeadManipulator.InterpolatedSpeed.Read(I_Adaptio.WeldHeadManipulator.InterpolatedSpeed);
    AdaptioIo.FromAdaptio.WeldHeadManipulator.XSpeed.Read(I_Adaptio.WeldHeadManipulator.XSpeed);
    AdaptioIo.FromAdaptio.WeldHeadManipulator.YSpeed.Read(I_Adaptio.WeldHeadManipulator.YSpeed);

    AdaptioIo.ToAdaptio.SystemVersions.Major.Write(Q_Adaptio.SystemVersions.Major);
    AdaptioIo.ToAdaptio.SystemVersions.Minor.Write(Q_Adaptio.SystemVersions.Minor);
    AdaptioIo.ToAdaptio.SystemVersions.Patch.Write(Q_Adaptio.SystemVersions.Patch);

    AdaptioIo.ToAdaptio.SystemControl.StartRequest.Write(Q_Adaptio.SystemControl.StartRequest);
    AdaptioIo.ToAdaptio.SystemControl.StopRequest.Write(Q_Adaptio.SystemControl.StopRequest);
    AdaptioIo.ToAdaptio.SystemControl.QuickStopRequest.Write(Q_Adaptio.SystemControl.QuickStopRequest);
    AdaptioIo.ToAdaptio.SystemControl.ShutdownRequest.Write(Q_Adaptio.SystemControl.ShutdownRequest);
    AdaptioIo.ToAdaptio.SystemControl.Heartbeat.Write(Q_Adaptio.SystemControl.Heartbeat);

    AdaptioIo.ToAdaptio.Joystick.State.Write(Q_Adaptio.Joystick.State);

    AdaptioIo.ToAdaptio.FluxSystem.State.Write(Q_Adaptio.FluxSystem.State);

    AdaptioIo.ToAdaptio.WeldControl.State.Write(Q_Adaptio.WeldControl.State);

    AdaptioIo.ToAdaptio.PowerSource1.Enabled.Write(Q_Adaptio.PowerSource1.Enabled);
    AdaptioIo.ToAdaptio.PowerSource1.State.Write(Q_Adaptio.PowerSource1.State);
    AdaptioIo.ToAdaptio.PowerSource1.ActiveVoltage.Write(Q_Adaptio.PowerSource1.ActiveVoltage);
    AdaptioIo.ToAdaptio.PowerSource1.ActiveCurrent.Write(Q_Adaptio.PowerSource1.ActiveCurrent);
    AdaptioIo.ToAdaptio.PowerSource1.ActiveWireSpeed.Write(Q_Adaptio.PowerSource1.ActiveWireSpeed);
    AdaptioIo.ToAdaptio.PowerSource1.ActiveRegulationType.Write(Q_Adaptio.PowerSource1.ActiveRegulationType);
    AdaptioIo.ToAdaptio.PowerSource1.ActiveWeldMethod.Write(Q_Adaptio.PowerSource1.ActiveWeldMethod);
    AdaptioIo.ToAdaptio.PowerSource1.ActiveAcFrequency.Write(Q_Adaptio.PowerSource1.ActiveAcFrequency);
    AdaptioIo.ToAdaptio.PowerSource1.ActiveAcBalance.Write(Q_Adaptio.PowerSource1.ActiveAcBalance);
    AdaptioIo.ToAdaptio.PowerSource1.ActiveAcOffset.Write(Q_Adaptio.PowerSource1.ActiveAcOffset);
    AdaptioIo.ToAdaptio.PowerSource1.ActiveAcPhaseShift.Write(Q_Adaptio.PowerSource1.ActiveAcPhaseShift);
    AdaptioIo.ToAdaptio.PowerSource1.ActiveStartAdjust.Write(Q_Adaptio.PowerSource1.ActiveStartAdjust);
    AdaptioIo.ToAdaptio.PowerSource1.ActiveRegulationDynamics.Write(Q_Adaptio.PowerSource1.ActiveRegulationDynamics);
    AdaptioIo.ToAdaptio.PowerSource1.ActiveRegulationInductance.Write(Q_Adaptio.PowerSource1.ActiveRegulationInductance);
    AdaptioIo.ToAdaptio.PowerSource1.ActiveIceWireSpeed.Write(Q_Adaptio.PowerSource1.ActiveIceWireSpeed);
    AdaptioIo.ToAdaptio.PowerSource1.MeasuredVoltage.Write(Q_Adaptio.PowerSource1.MeasuredVoltage);
    AdaptioIo.ToAdaptio.PowerSource1.MeasuredCurrent.Write(Q_Adaptio.PowerSource1.MeasuredCurrent);
    AdaptioIo.ToAdaptio.PowerSource1.MeasuredWireSpeed.Write(Q_Adaptio.PowerSource1.MeasuredWireSpeed);
    AdaptioIo.ToAdaptio.PowerSource1.MeasuredIceWireSpeed.Write(Q_Adaptio.PowerSource1.MeasuredIceWireSpeed);
    AdaptioIo.ToAdaptio.PowerSource1.CalculatedHeatInput.Write(Q_Adaptio.PowerSource1.CalculatedHeatInput);
    AdaptioIo.ToAdaptio.PowerSource1.CalculatedDepositionRate.Write(Q_Adaptio.PowerSource1.CalculatedDepositionRate);

    AdaptioIo.ToAdaptio.PowerSource2.Enabled.Write(Q_Adaptio.PowerSource2.Enabled);
    AdaptioIo.ToAdaptio.PowerSource2.State.Write(Q_Adaptio.PowerSource2.State);
    AdaptioIo.ToAdaptio.PowerSource2.ActiveVoltage.Write(Q_Adaptio.PowerSource2.ActiveVoltage);
    AdaptioIo.ToAdaptio.PowerSource2.ActiveCurrent.Write(Q_Adaptio.PowerSource2.ActiveCurrent);
    AdaptioIo.ToAdaptio.PowerSource2.ActiveWireSpeed.Write(Q_Adaptio.PowerSource2.ActiveWireSpeed);
    AdaptioIo.ToAdaptio.PowerSource2.ActiveRegulationType.Write(Q_Adaptio.PowerSource2.ActiveRegulationType);
    AdaptioIo.ToAdaptio.PowerSource2.ActiveWeldMethod.Write(Q_Adaptio.PowerSource2.ActiveWeldMethod);
    AdaptioIo.ToAdaptio.PowerSource2.ActiveAcFrequency.Write(Q_Adaptio.PowerSource2.ActiveAcFrequency);
    AdaptioIo.ToAdaptio.PowerSource2.ActiveAcBalance.Write(Q_Adaptio.PowerSource2.ActiveAcBalance);
    AdaptioIo.ToAdaptio.PowerSource2.ActiveAcOffset.Write(Q_Adaptio.PowerSource2.ActiveAcOffset);
    AdaptioIo.ToAdaptio.PowerSource2.ActiveAcPhaseShift.Write(Q_Adaptio.PowerSource2.ActiveAcPhaseShift);
    AdaptioIo.ToAdaptio.PowerSource2.ActiveStartAdjust.Write(Q_Adaptio.PowerSource2.ActiveStartAdjust);
    AdaptioIo.ToAdaptio.PowerSource2.ActiveRegulationDynamics.Write(Q_Adaptio.PowerSource2.ActiveRegulationDynamics);
    AdaptioIo.ToAdaptio.PowerSource2.ActiveRegulationInductance.Write(Q_Adaptio.PowerSource2.ActiveRegulationInductance);
    AdaptioIo.ToAdaptio.PowerSource2.ActiveIceWireSpeed.Write(Q_Adaptio.PowerSource2.ActiveIceWireSpeed);
    AdaptioIo.ToAdaptio.PowerSource2.MeasuredVoltage.Write(Q_Adaptio.PowerSource2.MeasuredVoltage);
    AdaptioIo.ToAdaptio.PowerSource2.MeasuredCurrent.Write(Q_Adaptio.PowerSource2.MeasuredCurrent);
    AdaptioIo.ToAdaptio.PowerSource2.MeasuredWireSpeed.Write(Q_Adaptio.PowerSource2.MeasuredWireSpeed);
    AdaptioIo.ToAdaptio.PowerSource2.MeasuredIceWireSpeed.Write(Q_Adaptio.PowerSource2.MeasuredIceWireSpeed);
    AdaptioIo.ToAdaptio.PowerSource2.CalculatedHeatInput.Write(Q_Adaptio.PowerSource2.CalculatedHeatInput);
    AdaptioIo.ToAdaptio.PowerSource2.CalculatedDepositionRate.Write(Q_Adaptio.PowerSource2.CalculatedDepositionRate);

    AdaptioIo.ToAdaptio.WeldAxis.InPosition.Write(Q_Adaptio.WeldAxis.InPosition);
    AdaptioIo.ToAdaptio.WeldAxis.ReferenceValid.Write(Q_Adaptio.WeldAxis.ReferenceValid);
    AdaptioIo.ToAdaptio.WeldAxis.State.Write(Q_Adaptio.WeldAxis.State);
    AdaptioIo.ToAdaptio.WeldAxis.ErrorCode.Write(Q_Adaptio.WeldAxis.ErrorCode);
    AdaptioIo.ToAdaptio.WeldAxis.AxisType.Write(Q_Adaptio.WeldAxis.AxisType);
    AdaptioIo.ToAdaptio.WeldAxis.Radius.Write(Q_Adaptio.WeldAxis.Radius);
    AdaptioIo.ToAdaptio.WeldAxis.Position.Write(Q_Adaptio.WeldAxis.Position);
    AdaptioIo.ToAdaptio.WeldAxis.LinearObjectDistance.Write(Q_Adaptio.WeldAxis.LinearObjectDistance);
    AdaptioIo.ToAdaptio.WeldAxis.Velocity.Write(Q_Adaptio.WeldAxis.Velocity);

    AdaptioIo.ToAdaptio.WeldHeadManipulator.InPosition.Write(Q_Adaptio.WeldHeadManipulator.InPosition);
    AdaptioIo.ToAdaptio.WeldHeadManipulator.State.Write(Q_Adaptio.WeldHeadManipulator.State);
    AdaptioIo.ToAdaptio.WeldHeadManipulator.XPosition.Write(Q_Adaptio.WeldHeadManipulator.XPosition);
    AdaptioIo.ToAdaptio.WeldHeadManipulator.YPosition.Write(Q_Adaptio.WeldHeadManipulator.YPosition);
    AdaptioIo.ToAdaptio.WeldHeadManipulator.InterpolatedSpeed.Write(Q_Adaptio.WeldHeadManipulator.InterpolatedSpeed);
    AdaptioIo.ToAdaptio.WeldHeadManipulator.XVelocity.Write(Q_Adaptio.WeldHeadManipulator.XVelocity);
    AdaptioIo.ToAdaptio.WeldHeadManipulator.YVelocity.Write(Q_Adaptio.WeldHeadManipulator.YVelocity);
END_PROGRAM

(* ---- BigBagFluxSystem.st ---- *)
USING Esab.WeldSystem.Flux;
Using Esab.Utils.Alarming;
Using Esab.Utils.Assets;

USING Siemens.Simatic.S71500.Tasks;
USING Siemens.Simatic.S71500.Alarming;

CONFIGURATION BigBagFluxSystemConfiguration

    TASK BigBagFluxSystemIoTask : ProgramCycle;

    PROGRAM BigBagFluxSystemIoReadWrite WITH BigBagFluxSystemIoTask: BigBagFluxSystemIoReadWrite;

    // Constants
    VAR_GLOBAL CONSTANT
    END_VAR

    // Objects
    VAR_GLOBAL
        {S7.Extern=Read}
        FluxSystem : BigBag.FluxSystem;
    END_VAR

    // Alarms
    VAR_GLOBAL
        BigBagErrorAlarmWrapper : AlarmWrapper;
        {S7.Alarm = NoAck, "Flux system (Big Bag): General error."}
        BigBagErrorAlarm : ProgramAlarm;

        BigBagSetupAlarmWrapper : AlarmWrapper;
        {S7.Alarm = NoAck, "Flux system (Big Bag): Setup error."}
        BigBagSetupAlarm : ProgramAlarm;
    END_VAR

    // Interface
    VAR_GLOBAL
        {S7.Extern=ReadWrite}
        FluxSystemIo : BigBag.Io;
    END_VAR
END_CONFIGURATION

FUNCTION InitializeBigBagFluxSystem
    VAR_INPUT
        Assets : IAssetsManager;
    END_VAR

    VAR_EXTERNAL
        FluxSystemIo : BigBag.Io;

        FluxSystem : BigBag.FluxSystem;

        BigBagErrorAlarmWrapper : AlarmWrapper;
        BigBagErrorAlarm : ProgramAlarm;
        BigBagSetupAlarmWrapper : AlarmWrapper;
        BigBagSetupAlarm : ProgramAlarm;
    END_VAR

    FluxSystemIo.Input.Temperature.Scale := REAL#0.1;

    BigBagErrorAlarmWrapper.Setup(REF(BigBagErrorAlarm));
    BigBagSetupAlarmWrapper.Setup(REF(BigBagSetupAlarm));
    FluxSystem.Setup(REF(FluxSystemIo), BigBagErrorAlarmWrapper, BigBagSetupAlarmWrapper);

    FluxSystem.SetIdentifier(Esab.AssetIdentifier#FluxSystem);
    Assets.RegisterAsset(REF(FluxSystem));
END_FUNCTION

PROGRAM BigBagFluxSystemIoReadWrite
    VAR_EXTERNAL
        FluxSystemIo : BigBag.Io;
        DI_B_FluxSystem_Error : BOOL;

        DQ_H_FluxSystem_Recover : BOOL;
        DQ_H_FluxSystem_Release : BOOL;
        AI_B_FluxSystem_Temperature : INT;
    END_VAR

    FluxSystemIo.Input.BigBagError.Read(DI_B_FluxSystem_Error);
    FluxSystemIo.Input.Temperature.Read(AI_B_FluxSystem_Temperature);

    FluxSystemIo.Output.Release.Write(DQ_H_FluxSystem_Release);
    FluxSystemIo.Output.Recover.Write(DQ_H_FluxSystem_Recover);
END_PROGRAM

(* ---- C_Hmi.st ---- *)
USING Esab.Hmi;
USING Esab.Utils.Timer;
USING Esab.Hmi.Modules;
Using Esab.Utils.Alarming;
USING Esab.Utils.Assets;

USING Siemens.Simatic.S71500.Tasks;
USING Siemens.Simatic.S71500.Alarming;

CONFIGURATION C_Hmi_Configuration

    TASK C_Hmi_IoTask : ProgramCycle;

    PROGRAM C_Hmi_IoReadWrite WITH C_Hmi_IoTask: C_Hmi_IoReadWrite;

    // Constants
    VAR_GLOBAL CONSTANT
    END_VAR

    // Objects
    VAR_GLOBAL
        C_Hmi : C_Hmi;
        C_EmergencyStop_Reset : PushButton;
        C_FluxSystem_Release : PushButton;
        C_HighSpeed : PushButton;
        C_WireFeed1 : TwinPushButton;
        C_WireFeed2 : TwinPushButton;
        C_WireFeed3 : TwinPushButton;
        C_TrackingOff : PushButton;
        C_MotionJoystick : DiscreteJoystick;
        C_MotionJoystick_LongHoldTimer : OnDelay;
        C_Tilt : TwinPushButton;
    END_VAR

    // Alarms
    VAR_GLOBAL
        C_Hmi_SetupAlarmWrapper : AlarmWrapper;
        {S7.Alarm = NoAck, "C HMI: Setup error."}
        C_Hmi_SetupAlarm : ProgramAlarm;
    END_VAR

    // Interface
    VAR_GLOBAL
        {S7.Extern=ReadWrite}
        C_Io_EmergencyStop_Reset : PushButtonIo;
        {S7.Extern=ReadWrite}
        C_Io_FluxSystem_Release : PushButtonIo;
        {S7.Extern=ReadWrite}
        C_Io_HighSpeed : PushButtonIo;
        {S7.Extern=ReadWrite}
        C_Io_WireFeed1 : TwinPushButtonIo;
        {S7.Extern=ReadWrite}
        C_Io_WireFeed2 : TwinPushButtonIo;
        {S7.Extern=ReadWrite}
        C_Io_WireFeed3 : TwinPushButtonIo;
        {S7.Extern=ReadWrite}
        C_Io_TrackingOff : PushButtonIo;
        {S7.Extern=ReadWrite}
        C_Io_MotionJoystick : DiscreteJoystickIo;
        {S7.Extern=ReadWrite}
        C_Io_Tilt : TwinPushButtonIo;
    END_VAR
END_CONFIGURATION

FUNCTION InitializeC
    VAR_INPUT
        assetsManager : IAssetsManager;
    END_VAR

    VAR_EXTERNAL
        C_Hmi : C_Hmi;
        C_EmergencyStop_Reset : PushButton;
        C_FluxSystem_Release : PushButton;
        C_HighSpeed : PushButton;
        C_WireFeed1 : TwinPushButton;
        C_WireFeed2 : TwinPushButton;
        C_WireFeed3 : TwinPushButton;
        C_TrackingOff : PushButton;
        C_MotionJoystick : DiscreteJoystick;
        C_MotionJoystick_LongHoldTimer : OnDelay;
        C_Tilt : TwinPushButton;

        C_Io_EmergencyStop_Reset : PushButtonIo;
        C_Io_FluxSystem_Release : PushButtonIo;
        C_Io_HighSpeed : PushButtonIo;
        C_Io_WireFeed1 : TwinPushButtonIo;
        C_Io_WireFeed2 : TwinPushButtonIo;
        C_Io_WireFeed3 : TwinPushButtonIo;
        C_Io_TrackingOff : PushButtonIo;
        C_Io_MotionJoystick : DiscreteJoystickIo;
        C_Io_Tilt : TwinPushButtonIo;

        C_Hmi_SetupAlarmWrapper : AlarmWrapper;
        C_Hmi_SetupAlarm : ProgramAlarm;
    END_VAR

    C_EmergencyStop_Reset.Setup(io := REF(C_Io_EmergencyStop_Reset));
    C_EmergencyStop_Reset.SetIdentifier(Esab.AssetIdentifier#C_PushButton_EmergencyStop_Reset);
    assetsManager.RegisterAsset(REF(C_EmergencyStop_Reset));

    C_FluxSystem_Release.Setup(io := REF(C_Io_FluxSystem_Release));
    C_FluxSystem_Release.SetIdentifier(Esab.AssetIdentifier#C_PushButton_FluxSystem_Release);
    assetsManager.RegisterAsset(REF(C_FluxSystem_Release));

    C_HighSpeed.Setup(io := REF(C_Io_HighSpeed));
    C_HighSpeed.SetIdentifier(Esab.AssetIdentifier#C_PushButton_System_HighSpeed);
    assetsManager.RegisterAsset(REF(C_HighSpeed));

    C_WireFeed1.Setup(io := REF(C_Io_WireFeed1));
    C_WireFeed1.SetIdentifier(Esab.AssetIdentifier#C_TwinPushButton_WireFeed1);
    assetsManager.RegisterAsset(REF(C_WireFeed1));

    C_WireFeed2.Setup(io := REF(C_Io_WireFeed2));
    C_WireFeed2.SetIdentifier(Esab.AssetIdentifier#C_TwinPushButton_WireFeed2);
    assetsManager.RegisterAsset(REF(C_WireFeed2));

    C_WireFeed3.Setup(io := REF(C_Io_WireFeed3));
    C_WireFeed3.SetIdentifier(Esab.AssetIdentifier#C_TwinPushButton_WireFeed3);
    assetsManager.RegisterAsset(REF(C_WireFeed3));

    C_TrackingOff.Setup(io := REF(C_Io_TrackingOff));
    C_TrackingOff.SetIdentifier(Esab.AssetIdentifier#C_PushButton_TrackingOff);
    assetsManager.RegisterAsset(REF(C_TrackingOff));

    C_MotionJoystick.Setup(io := REF(C_Io_MotionJoystick), longHoldTimer := C_MotionJoystick_LongHoldTimer);
    C_MotionJoystick.SetIdentifier(Esab.AssetIdentifier#C_Joystick_MotionJoystick);
    assetsManager.RegisterAsset(REF(C_MotionJoystick));

    C_Hmi_SetupAlarmWrapper.Setup(REF(C_Hmi_SetupAlarm));

    C_Hmi.Setup(assetsManager, C_Hmi_SetupAlarmWrapper);
END_FUNCTION

PROGRAM C_Hmi_IoReadWrite
    VAR_EXTERNAL
        C_Io_EmergencyStop_Reset : PushButtonIo;
        C_Io_FluxSystem_Release : PushButtonIo;
        C_Io_HighSpeed : PushButtonIo;
        C_Io_WireFeed1 : TwinPushButtonIo;
        C_Io_WireFeed2 : TwinPushButtonIo;
        C_Io_WireFeed3 : TwinPushButtonIo;
        C_Io_TrackingOff : PushButtonIo;
        C_Io_MotionJoystick : DiscreteJoystickIo;
        C_Io_Tilt : TwinPushButtonIo;

        DI_C_PushButton_EmergencyStop_Reset : BOOL;
        DQ_C_PushButton_EmergencyStop_Reset : BOOL;

        DI_C_PushButton_FluxSystem_Release : BOOL;
        DQ_C_PushButton_FluxSystem_Release : BOOL;

        DI_C_PushButton_HighSpeed : BOOL;
        DQ_C_PushButton_HighSpeed : BOOL;

        DI_C_PushButton_WireFeed1_Up : BOOL;
        DI_C_PushButton_WireFeed1_Down : BOOL;

        DI_C_PushButton_WireFeed2_Up : BOOL;
        DI_C_PushButton_WireFeed2_Down : BOOL;

        DI_C_PushButton_WireFeed3_Up : BOOL;
        DI_C_PushButton_WireFeed3_Down : BOOL;

        DI_C_PushButton_TrackingOff : BOOL;
        DQ_C_PushButton_TrackingOff : BOOL;

        DI_C_MotionJoystick_Up : BOOL;
        DI_C_MotionJoystick_Down : BOOL;
        DI_C_MotionJoystick_Triangle : BOOL;
        DI_C_MotionJoystick_Square : BOOL;

        DI_C_PushButton_Tilt_Left : BOOL;
        DI_C_PushButton_Tilt_Right : BOOL;
    END_VAR

    C_Io_EmergencyStop_Reset.Pressed.Read(DI_C_PushButton_EmergencyStop_Reset);
    C_Io_EmergencyStop_Reset.Status.Write(DQ_C_PushButton_EmergencyStop_Reset);

    C_Io_FluxSystem_Release.Pressed.Read(DI_C_PushButton_FluxSystem_Release);
    C_Io_FluxSystem_Release.Status.Write(DQ_C_PushButton_FluxSystem_Release);

    C_Io_HighSpeed.Pressed.Read(DI_C_PushButton_HighSpeed);
    C_Io_HighSpeed.Status.Write(DQ_C_PushButton_HighSpeed);

    C_Io_WireFeed1.Direction1.Read(DI_C_PushButton_WireFeed1_Up);
    C_Io_WireFeed1.Direction2.Read(DI_C_PushButton_WireFeed1_Down);

    C_Io_WireFeed2.Direction1.Read(DI_C_PushButton_WireFeed2_Up);
    C_Io_WireFeed2.Direction2.Read(DI_C_PushButton_WireFeed2_Down);

    C_Io_WireFeed3.Direction1.Read(DI_C_PushButton_WireFeed3_Up);
    C_Io_WireFeed3.Direction2.Read(DI_C_PushButton_WireFeed3_Down);

    C_Io_TrackingOff.Pressed.Read(DI_C_PushButton_TrackingOff);
    C_Io_TrackingOff.Status.Write(DQ_C_PushButton_TrackingOff);

    C_Io_MotionJoystick.Up.Read(DI_C_MotionJoystick_Up);
    C_Io_MotionJoystick.Down.Read(DI_C_MotionJoystick_Down);
    C_Io_MotionJoystick.Triangle.Read(DI_C_MotionJoystick_Triangle);
    C_Io_MotionJoystick.Square.Read(DI_C_MotionJoystick_Square);

    C_Io_Tilt.Direction1.Read(DI_C_PushButton_Tilt_Left);
    C_Io_Tilt.Direction2.Read(DI_C_PushButton_Tilt_Right);
END_PROGRAM

(* ---- EmergencyStopCircuit.st ---- *)
USING Esab.Hmi;
USING Esab.Utils.Timer;
USING Esab.Hmi.Modules;
USING Esab.Utils.Assets;
USING Esab.Utils.EmergencyStop;

USING Siemens.Simatic.S71500.Tasks;

CONFIGURATION EmergencyStopCircuit_Configuration

    TASK EmergencyStopCircuit_IoTask : ProgramCycle;

    PROGRAM EmergencyStopCircuit_IoReadWrite WITH EmergencyStopCircuit_IoTask: EmergencyStopCircuit_IoReadWrite;

    // Constants
    VAR_GLOBAL CONSTANT
    END_VAR

    // Objects
    VAR_GLOBAL
        EmergencyStopCircuit : EmergencyStopCircuit;
    END_VAR

    // Interface
    VAR_GLOBAL
        {S7.Extern=ReadWrite}
        EmergencyStopCircuitIo : EmergencyStopCircuitIo;
    END_VAR
END_CONFIGURATION

FUNCTION InitializeEmergencyStopCircuit
    VAR_INPUT
        Assets : IAssetsManager;
    END_VAR

    VAR_EXTERNAL
        EmergencyStopCircuit : EmergencyStopCircuit;
        EmergencyStopCircuitIo : EmergencyStopCircuitIo;
    END_VAR

    EmergencyStopCircuit.Io := REF(EmergencyStopCircuitIo);
    EmergencyStopCircuit.SetIdentifier(Esab.AssetIdentifier#EmergencyStopCircuit);
    Assets.RegisterAsset(REF(EmergencyStopCircuit));
END_FUNCTION

PROGRAM EmergencyStopCircuit_IoReadWrite
    VAR_EXTERNAL
        EmergencyStopCircuitIo : EmergencyStopCircuitIo;

        DI_B_System_EmergencyStop_OK : BOOL;
    END_VAR

    EmergencyStopCircuitIo.LoopClosed.Read(DI_B_System_EmergencyStop_OK);
END_PROGRAM

(* ---- P_Hmi.st ---- *)
USING Esab.Hmi;
USING Esab.Utils.Timer;
USING Esab.Hmi.Modules;
Using Esab.Utils.Alarming;
USING Esab.Utils.Assets;

USING Siemens.Simatic.S71500.Tasks;
USING Siemens.Simatic.S71500.Alarming;

CONFIGURATION P_Hmi_Configuration

    TASK P_Hmi_IoTask : ProgramCycle;

    PROGRAM P_Hmi_IoReadWrite WITH P_Hmi_IoTask: P_Hmi_IoReadWrite;

    // Constants
    VAR_GLOBAL CONSTANT
    END_VAR

    // Objects
    VAR_GLOBAL
        P_Hmi : P_Hmi;
        P_EmergencyStop_Reset : PushButton;
        P_FluxSystem_Release : PushButton;
        P_FluxSystem_Recover : PushButton;
        P_HighSpeedButton : PushButton;
        P_WireFeed1 : TwinPushButton;
        P_WireFeed2 : TwinPushButton;
        P_MotionJoystick_AxisSelection : PushButton;
        P_MotionJoystick : DiscreteJoystick;
        P_MotionJoystick_LongHoldTimer : OnDelay;
        P_AxisJog_AxisSelection : PushButton;
        P_AxisJog : TwinPushButton;
        P_Start : PushButton;
        P_Stop : PushButton;
    END_VAR

    // Alarms
    VAR_GLOBAL
        P_Hmi_SetupAlarmWrapper : AlarmWrapper;
        {S7.Alarm = NoAck, "P HMI: Setup error."}
        P_Hmi_SetupAlarm : ProgramAlarm;
    END_VAR

    // Interface
    VAR_GLOBAL
        {S7.Extern=ReadWrite}
        P_Io_EmergencyStop_Reset : PushButtonIo;
        {S7.Extern=ReadWrite}
        P_Io_FluxSystem_Release : PushButtonIo;
        {S7.Extern=ReadWrite}
        P_Io_FluxSystem_Recover : PushButtonIo;
        {S7.Extern=ReadWrite}
        P_Io_WireFeed1 : TwinPushButtonIo;
        {S7.Extern=ReadWrite}
        P_Io_WireFeed2 : TwinPushButtonIo;
        {S7.Extern=ReadWrite}
        P_Io_HighSpeedButton : PushButtonIo;
        {S7.Extern=ReadWrite}
        P_Io_MotionJoystick_AxisSelection : PushButtonIo;
        {S7.Extern=ReadWrite}
        P_Io_MotionJoystick : DiscreteJoystickIo;
        {S7.Extern=ReadWrite}
        P_Io_AxisJog_AxisSelection : PushButtonIo;
        {S7.Extern=ReadWrite}
        P_Io_AxisJog : TwinPushButtonIo;
        {S7.Extern=ReadWrite}
        P_Io_Start : PushButtonIo;
        {S7.Extern=ReadWrite}
        P_Io_Stop : PushButtonIo;
    END_VAR
END_CONFIGURATION

FUNCTION InitializeP
    VAR_INPUT
        assetsManager : IAssetsManager;
    END_VAR

    VAR_EXTERNAL
        P_Hmi : P_Hmi;
        P_EmergencyStop_Reset : PushButton;
        P_FluxSystem_Release : PushButton;
        P_FluxSystem_Recover : PushButton;
        P_HighSpeedButton : PushButton;
        P_WireFeed1 : TwinPushButton;
        P_WireFeed2 : TwinPushButton;
        P_MotionJoystick_AxisSelection : PushButton;
        P_MotionJoystick : DiscreteJoystick;
        P_MotionJoystick_LongHoldTimer : OnDelay;
        P_AxisJog_AxisSelection : PushButton;
        P_AxisJog : TwinPushButton;
        P_Start : PushButton;
        P_Stop : PushButton;

        P_Io_EmergencyStop_Reset : PushButtonIo;
        P_Io_FluxSystem_Release : PushButtonIo;
        P_Io_FluxSystem_Recover : PushButtonIo;
        P_Io_WireFeed1 : TwinPushButtonIo;
        P_Io_WireFeed2 : TwinPushButtonIo;
        P_Io_HighSpeedButton : PushButtonIo;
        P_Io_MotionJoystick_AxisSelection : PushButtonIo;
        P_Io_MotionJoystick : DiscreteJoystickIo;
        P_Io_AxisJog_AxisSelection : PushButtonIo;
        P_Io_AxisJog : TwinPushButtonIo;
        P_Io_Start : PushButtonIo;
        P_Io_Stop : PushButtonIo;

        P_Hmi_SetupAlarmWrapper : AlarmWrapper;
        P_Hmi_SetupAlarm : ProgramAlarm;
    END_VAR

    P_EmergencyStop_Reset.Setup(io := REF(P_Io_EmergencyStop_Reset));
    P_EmergencyStop_Reset.SetIdentifier(Esab.AssetIdentifier#P_PushButton_EmergencyStop_Reset);
    assetsManager.RegisterAsset(REF(P_EmergencyStop_Reset));

    P_FluxSystem_Release.Setup(io := REF(P_Io_FluxSystem_Release));
    P_FluxSystem_Release.SetIdentifier(Esab.AssetIdentifier#P_PushButton_FluxSystem_Release);
    assetsManager.RegisterAsset(REF(P_FluxSystem_Release));

    P_FluxSystem_Recover.Setup(io := REF(P_Io_FluxSystem_Recover));
    P_FluxSystem_Recover.SetIdentifier(Esab.AssetIdentifier#P_PushButton_FluxSystem_Recover);
    assetsManager.RegisterAsset(REF(P_FluxSystem_Recover));

    P_HighSpeedButton.Setup(io := REF(P_Io_HighSpeedButton));
    P_HighSpeedButton.SetIdentifier(Esab.AssetIdentifier#P_PushButton_System_HighSpeed);
    assetsManager.RegisterAsset(REF(P_HighSpeedButton));

    P_WireFeed1.Setup(io := REF(P_Io_WireFeed1));
    P_WireFeed1.SetIdentifier(Esab.AssetIdentifier#P_TwinPushButton_WireFeed1);
    assetsManager.RegisterAsset(REF(P_WireFeed1));

    P_WireFeed2.Setup(io := REF(P_Io_WireFeed2));
    P_WireFeed2.SetIdentifier(Esab.AssetIdentifier#P_TwinPushButton_WireFeed2);
    assetsManager.RegisterAsset(REF(P_WireFeed2));

    P_MotionJoystick_AxisSelection.Setup(io := REF(P_Io_MotionJoystick_AxisSelection));
    P_MotionJoystick_AxisSelection.SetIdentifier(Esab.AssetIdentifier#P_PushButton_MotionJoystick_AxisSelection);
    assetsManager.RegisterAsset(REF(P_MotionJoystick_AxisSelection));

    P_MotionJoystick.Setup(io := REF(P_Io_MotionJoystick), longHoldTimer := P_MotionJoystick_LongHoldTimer);
    P_MotionJoystick.SetIdentifier(Esab.AssetIdentifier#P_Joystick_MotionJoystick);
    assetsManager.RegisterAsset(REF(P_MotionJoystick));

    P_AxisJog_AxisSelection.Setup(io := REF(P_Io_AxisJog_AxisSelection));
    P_AxisJog_AxisSelection.SetIdentifier(Esab.AssetIdentifier#P_PushButton_AxisJog_AxisSelection);
    assetsManager.RegisterAsset(REF(P_AxisJog_AxisSelection));

    P_AxisJog.Setup(io := REF(P_Io_AxisJog));
    P_AxisJog.SetIdentifier(Esab.AssetIdentifier#P_TwinPushButton_AxisJog);
    assetsManager.RegisterAsset(REF(P_AxisJog));

    P_Start.Setup(io := REF(P_Io_Start));
    P_Start.SetIdentifier(Esab.AssetIdentifier#P_PushButton_Start);
    assetsManager.RegisterAsset(REF(P_Start));

    P_Stop.Setup(io := REF(P_Io_Stop));
    P_Stop.SetIdentifier(Esab.AssetIdentifier#P_PushButton_Stop);
    assetsManager.RegisterAsset(REF(P_Stop));

    P_Hmi_SetupAlarmWrapper.Setup(REF(P_Hmi_SetupAlarm));

    P_Hmi.Setup(assetsManager, P_Hmi_SetupAlarmWrapper);
END_FUNCTION

PROGRAM P_Hmi_IoReadWrite
    VAR_EXTERNAL
        P_Io_EmergencyStop_Reset : PushButtonIo;
        P_Io_FluxSystem_Release : PushButtonIo;
        P_Io_FluxSystem_Recover : PushButtonIo;
        P_Io_WireFeed1 : TwinPushButtonIo;
        P_Io_WireFeed2 : TwinPushButtonIo;
        P_Io_HighSpeedButton : PushButtonIo;
        P_Io_MotionJoystick_AxisSelection : PushButtonIo;
        P_Io_MotionJoystick : DiscreteJoystickIo;
        P_Io_AxisJog_AxisSelection : PushButtonIo;
        P_Io_AxisJog : TwinPushButtonIo;
        P_Io_Start : PushButtonIo;
        P_Io_Stop : PushButtonIo;

        DI_P_PushButton_EmergencyStop_Reset : BOOL;
        DQ_P_PushButton_EmergencyStop_Reset : BOOL;

        DI_P_PushButton_FluxSystem_Release : BOOL;
        DQ_P_PushButton_FluxSystem_Release : BOOL;

        DI_P_PushButton_FluxSystem_Recover : BOOL;
        DQ_P_PushButton_FluxSystem_Recover : BOOL;

        DI_P_PushButton_HighSpeed : BOOL;
        DQ_P_PushButton_HighSpeed : BOOL;

        DI_P_PushButton_WireFeed1_Up : BOOL;
        DI_P_PushButton_WireFeed1_Down : BOOL;

        DI_P_PushButton_WireFeed2_Up : BOOL;
        DI_P_PushButton_WireFeed2_Down : BOOL;

        DI_P_MotionJoystick_AxisSelection : BOOL;
        DQ_P_MotionJoystick_AxisSelection : BOOL;
        DI_P_MotionJoystick_Up : BOOL;
        DI_P_MotionJoystick_Down : BOOL;
        DI_P_MotionJoystick_Triangle : BOOL;
        DI_P_MotionJoystick_Square : BOOL;

        DI_P_PushButton_AxisJog_AxisSelection : BOOL;
        DQ_P_PushButton_AxisJog_AxisSelection : BOOL;

        DI_P_PushButton_AxisJog_Triangle : BOOL;
        DI_P_PushButton_AxisJog_Square : BOOL;

        DI_P_PushButton_Start : BOOL;
        DQ_P_PushButton_Start : BOOL;

        DI_P_PushButton_Stop : BOOL;
        DQ_P_PushButton_Stop : BOOL;
    END_VAR

    P_Io_EmergencyStop_Reset.Pressed.Read(DI_P_PushButton_EmergencyStop_Reset);
    P_Io_EmergencyStop_Reset.Status.Write(DQ_P_PushButton_EmergencyStop_Reset);

    P_Io_FluxSystem_Release.Pressed.Read(DI_P_PushButton_FluxSystem_Release);
    P_Io_FluxSystem_Release.Status.Write(DQ_P_PushButton_FluxSystem_Release);

    P_Io_FluxSystem_Recover.Pressed.Read(DI_P_PushButton_FluxSystem_Recover);
    P_Io_FluxSystem_Recover.Status.Write(DQ_P_PushButton_FluxSystem_Recover);

    P_Io_HighSpeedButton.Pressed.Read(DI_P_PushButton_HighSpeed);
    P_Io_HighSpeedButton.Status.Write(DQ_P_PushButton_HighSpeed);

    P_Io_WireFeed1.Direction1.Read(DI_P_PushButton_WireFeed1_Up);
    P_Io_WireFeed1.Direction2.Read(DI_P_PushButton_WireFeed1_Down);

    P_Io_WireFeed2.Direction1.Read(DI_P_PushButton_WireFeed2_Up);
    P_Io_WireFeed2.Direction2.Read(DI_P_PushButton_WireFeed2_Down);

    P_Io_MotionJoystick_AxisSelection.Pressed.Read(DI_P_MotionJoystick_AxisSelection);
    P_Io_MotionJoystick_AxisSelection.Status.Write(DQ_P_MotionJoystick_AxisSelection);

    P_Io_MotionJoystick.Up.Read(DI_P_MotionJoystick_Up);
    P_Io_MotionJoystick.Down.Read(DI_P_MotionJoystick_Down);
    P_Io_MotionJoystick.Triangle.Read(DI_P_MotionJoystick_Triangle);
    P_Io_MotionJoystick.Square.Read(DI_P_MotionJoystick_Square);

    P_Io_AxisJog_AxisSelection.Pressed.Read(DI_P_MotionJoystick_AxisSelection);
    P_Io_AxisJog_AxisSelection.Status.Write(DQ_P_MotionJoystick_AxisSelection);

    P_Io_AxisJog.Direction1.Read(DI_P_PushButton_AxisJog_Triangle);
    P_Io_AxisJog.Direction2.Read(DI_P_PushButton_AxisJog_Square);

    P_Io_Start.Pressed.Read(DI_P_PushButton_Start);
    P_Io_Start.Status.Write(DQ_P_PushButton_Start);

    P_Io_Stop.Pressed.Read(DI_P_PushButton_Stop);
    P_Io_Stop.Status.Write(DQ_P_PushButton_Stop);
END_PROGRAM

(* ---- Platform.st ---- *)
USING Esab.Hmi;
USING Esab.Utils;
USING Esab.Utils.Assets;
USING Esab.Io;
USING Esab.Utils.Timer;
USING Esab.Platforms;
USING Esab.Hmi.Modules;

USING Siemens.Simatic.S71500.Tasks;

CONFIGURATION Platform
    TASK MainTask : ProgramCycle;
    TASK AwsStartup : Startup;

    PROGRAM MainProgram WITH MainTask: MainProgram;
    PROGRAM StartupProgram WITH AwsStartup : InitializeConfiguration;

    VAR_GLOBAL
        AssetsManager : AssetsManager;
    END_VAR

END_CONFIGURATION

/// This program is used to wire up I/O and other initialization to all the different objects.
PROGRAM InitializeConfiguration

    VAR_EXTERNAL
        AssetsManager : Esab.Utils.Assets.AssetsManager;
    END_VAR

    InitializeGlobalState(AssetsManager);
    InitializeWebApi(AssetsManager);
    InitializeP(AssetsManager);
    InitializeC(AssetsManager);
    InitializeEmergencyStopCircuit(AssetsManager);
    InitializeRollerBed(AssetsManager);
    InitializeBigBagFluxSystem(AssetsManager);
    InitializePs1(AssetsManager);
    InitializePs2(AssetsManager);
    InitializeSlideCrossAxis(AssetsManager);
    InitializeMultiWeldSystem(AssetsManager);
    InitializeAdaptio(AssetsManager);
    InitializeWeldHeadManipulator(AssetsManager);
    InitializeUps(AssetsManager);
END_PROGRAM

PROGRAM MainProgram
    VAR_EXTERNAL
        AssetsManager : AssetsManager;
        WebApi : Esab.Api.WebApi;
        P_Hmi : Esab.Hmi.P_Hmi;
        C_Hmi : Esab.Hmi.C_Hmi;
        Adaptio : Esab.Modes.Adaptio;
    END_VAR

    AssetsManager.Execute();

    Adaptio.Execute();
    WebApi.Execute();
    P_Hmi.Execute();
    C_Hmi.Execute();
END_PROGRAM

(* ---- PointLaser.st ---- *)
USING Esab.Peripheral;
Using Esab.Utils.Alarming;
Using Esab.Utils.Assets;

USING Siemens.Simatic.S71500.Tasks;
USING Siemens.Simatic.S71500.Alarming;

CONFIGURATION PointLaserConfiguration

    TASK PointLaserIoTask : ProgramCycle;

    PROGRAM PointLaserIoReadWrite WITH PointLaserIoTask: PointLaserIoReadWrite;

    // Constants
    VAR_GLOBAL CONSTANT
    END_VAR

    // Objects
    VAR_GLOBAL
        {S7.Extern=Read}
        PointLaser : ActivatableAsset;
    END_VAR

    // Alarms
    VAR_GLOBAL
        PointLaserSetupAlarmWrapper : AlarmWrapper;
        {S7.Alarm = NoAck, "Point laser: Setup error."}
        PointLaserSetupAlarm : ProgramAlarm;
    END_VAR

    // Interface
    VAR_GLOBAL
        {S7.Extern=ReadWrite}
        PointLaserIo : Io;
    END_VAR
END_CONFIGURATION

FUNCTION InitializePointLaser
    VAR_INPUT
        Assets : IAssetsManager;
    END_VAR

    VAR_EXTERNAL
        PointLaserIo : Io;
        PointLaser : ActivatableAsset;
        PointLaserSetupAlarmWrapper : AlarmWrapper;
        PointLaserSetupAlarm : ProgramAlarm;
    END_VAR

    PointLaserSetupAlarmWrapper.Setup(REF(PointLaserSetupAlarm));
    PointLaser.Setup(REF(PointLaserIo), PointLaserSetupAlarmWrapper);

    PointLaser.SetIdentifier(Esab.AssetIdentifier#PointLaser);
    Assets.RegisterAsset(REF(PointLaser));
END_FUNCTION

PROGRAM PointLaserIoReadWrite
    VAR_EXTERNAL
        PointLaserIo : Io;
        DQ_H_LaserPointer_Enable : BOOL;
    END_VAR

    PointLaserIo.Active.Write(DQ_H_LaserPointer_Enable);
END_PROGRAM

(* ---- PowerSource1.st ---- *)
USING Esab.WeldSystem.PowerSources;
USING Esab.WeldSystem;
USING Esab.Io;
USING Esab.Utils.Assets;
USING Esab.Utils.Timer;
Using Esab.Utils.Alarming;

USING Siemens.Simatic.S71500.Tasks;
USING Siemens.Simatic.S71500.Alarming;

CONFIGURATION PowerSource1Configuration

    TASK PowerSource1IoTask : ProgramCycle;

    PROGRAM PowerSource1IoProgram WITH PowerSource1IoTask: PowerSource1IoReadWrite;

    // Constants
    VAR_GLOBAL CONSTANT
        PAB1_HWID : WORD := WORD#261;
        PAB1_DEVID : WORD := WORD#262;
    END_VAR

    // Objects
    VAR_GLOBAL
        PowerSource1 : Aristo1000.PowerSource;
        Ps1HeartbeatTimer : OnDelay;
        Ps1Heartbeat : Heartbeat;
        Ps1AsyncInterface : AsyncInterface;
        Ps1AsyncReader : AsyncReader;
        Ps1AsyncWriter : AsyncWriter;
        Ps1AsyncCommands : AsyncCommands;
    END_VAR

    // Alarms
    VAR_GLOBAL
        // PS1 Alarms
        Ps1ErrorAlarmWrapper : AlarmWrapper;
        {S7.Alarm = NoAck, "Power source 1: Error."}
        Ps1ErrorAlarm : ProgramAlarm;

        Ps1HeartbeatAlarmWrapper : AlarmWrapper;
        {S7.Alarm = NoAck, "Power source 1: No heartbeat."}
        Ps1HeartbeatAlarm : ProgramAlarm;

        Ps1AsyncCommandReadAlarmWrapper : AlarmWrapper;
        {S7.Alarm = NoAck, "Power source 1: Async command (READ) @1%u@ failed."}
        Ps1AsyncCommandReadAlarm : ProgramAlarm;

        Ps1AsyncCommandWriteAlarmWrapper : AlarmWrapper;
        {S7.Alarm = NoAck, "Power source 1: Async command (WRITE) @1%u@ failed."}
        Ps1AsyncCommandWriteAlarm : ProgramAlarm;

        Ps1AsyncCommandNullAlarmWrapper : AlarmWrapper;
        {S7.Alarm = NoAck, "Power source 1: Async command response is NULL."}
        Ps1AsyncCommandNullAlarm : ProgramAlarm;

        Ps1SetupAlarmWrapper : AlarmWrapper;
        {S7.Alarm = NoAck, "Power source 1: Setup error."}
        Ps1SetupAlarm : ProgramAlarm;

        // Ps1 Async Interface Alarms
        Ps1InvalidCommandTypeAlarmWrapper : AlarmWrapper;
        {S7.Alarm = NoAck, "Power source 1: Async Interface: Invalid command type."}
        PS1InvalidCommandTypeAlarm : ProgramAlarm;

        Ps1PoppedNullCommandAlarmWrapper : AlarmWrapper;
        {S7.Alarm = NoAck, "Power source 1: Async Interface: The popped command is NULL."}
        Ps1PoppedNullCommandAlarm : ProgramAlarm;

        Ps1InvalidCommandAlarmWrapper : AlarmWrapper;
        {S7.Alarm = NoAck, "Power source 1: Async Interface: The type of the popped command is not AsyncCommand."}
        Ps1InvalidCommandAlarm : ProgramAlarm;

        // PS1 Async Reader Alarms
        Ps1AsyncReaderErrorAlarmWrapper : AlarmWrapper;
        {S7.Alarm = NoAck, "Power source 1: Async Reader: Error when reading async data, status: @1%u@."}
        Ps1AsyncReaderErrorAlarm : ProgramAlarm;

        // PS1 Async Writer Alarms
        Ps1AsyncWriterErrorAlarmWrapper : AlarmWrapper;
        {S7.Alarm = NoAck, "Power source 1: Async Writer: Error when writing async data, status: @1%u@."}
        Ps1AsyncWriterErrorAlarm : ProgramAlarm;
    END_VAR

    // Interface
    VAR_GLOBAL
        {S7.Extern=ReadWrite}
        PS1_Data : Io;
    END_VAR

    // Retain
    VAR_GLOBAL RETAIN
        Ps1RuntimeParameters : RuntimeParameters;
        Ps1HardwareConfiguration : HardwareConfiguration;
    END_VAR
END_CONFIGURATION

FUNCTION InitializePs1
    VAR_INPUT
        assetsManager : IAssetsManager;
    END_VAR

    VAR_EXTERNAL CONSTANT
        PAB1_HWID : WORD;
        PAB1_DEVID : WORD;
    END_VAR

    VAR_EXTERNAL
        PS1_Data : Io;

        PowerSource1 : Aristo1000.PowerSource;
        Ps1HeartbeatTimer : OnDelay;
        Ps1Heartbeat : Heartbeat;
        Ps1AsyncInterface : AsyncInterface;
        Ps1AsyncReader : AsyncReader;
        Ps1AsyncWriter : AsyncWriter;
        Ps1AsyncCommands : AsyncCommands;
        Ps1RuntimeParameters : RuntimeParameters;
        Ps1HardwareConfiguration : HardwareConfiguration;

        Ps1ErrorAlarmWrapper : AlarmWrapper;
        Ps1HeartbeatAlarmWrapper : AlarmWrapper;
        Ps1AsyncCommandReadAlarmWrapper : AlarmWrapper;
        Ps1AsyncCommandWriteAlarmWrapper : AlarmWrapper;
        Ps1AsyncCommandNullAlarmWrapper : AlarmWrapper;
        Ps1SetupAlarmWrapper : AlarmWrapper;

        Ps1ErrorAlarm : ProgramAlarm;
        Ps1HeartbeatAlarm : ProgramAlarm;
        Ps1AsyncCommandReadAlarm : ProgramAlarm;
        Ps1AsyncCommandWriteAlarm : ProgramAlarm;
        Ps1AsyncCommandNullAlarm : ProgramAlarm;
        Ps1SetupAlarm : ProgramAlarm;

        Ps1InvalidCommandTypeAlarmWrapper : AlarmWrapper;
        Ps1PoppedNullCommandAlarmWrapper : AlarmWrapper;
        Ps1InvalidCommandAlarmWrapper : AlarmWrapper;

        Ps1InvalidCommandTypeAlarm : ProgramAlarm;
        Ps1PoppedNullCommandAlarm : ProgramAlarm;
        Ps1InvalidCommandAlarm : ProgramAlarm;

        Ps1AsyncReaderErrorAlarmWrapper : AlarmWrapper;
        Ps1AsyncWriterErrorAlarmWrapper : AlarmWrapper;

        Ps1AsyncReaderErrorAlarm : ProgramAlarm;
        Ps1AsyncWriterErrorAlarm : ProgramAlarm;
    END_VAR

    // Setup heartbeat
    Ps1Heartbeat.Input := PS1_Data.Pab.Input.Heartbeat;
    Ps1Heartbeat.Timer := Ps1HeartbeatTimer;

    // Setup async interface
    Ps1AsyncReader.HwId := PAB1_HWID;
    Ps1AsyncWriter.HwId := PAB1_HWID;

    // Setup alarm wrappers
    Ps1ErrorAlarmWrapper.Setup(REF(Ps1ErrorAlarm));
    Ps1HeartbeatAlarmWrapper.Setup(REF(Ps1HeartbeatAlarm));
    Ps1AsyncCommandReadAlarmWrapper.Setup(REF(Ps1AsyncCommandReadAlarm));
    Ps1AsyncCommandWriteAlarmWrapper.Setup(REF(Ps1AsyncCommandWriteAlarm));
    Ps1AsyncCommandNullAlarmWrapper.Setup(REF(Ps1AsyncCommandNullAlarm));
    Ps1SetupAlarmWrapper.Setup(REF(Ps1SetupAlarm));

    // Setup PowerSource using Setup method
    PowerSource1.Setup(
        id := UINT#1,
        ioDeviceId := PAB1_DEVID,
        heartbeat := Ps1Heartbeat,
        io := REF(PS1_Data),
        runtimeParameters := REF(Ps1RuntimeParameters),
        hardwareConfiguration := REF(Ps1HardwareConfiguration),
        asyncInterface := Ps1AsyncInterface,
        errorAlarm := Ps1ErrorAlarmWrapper,
        heartbeatAlarm := Ps1HeartbeatAlarmWrapper,
        asyncCommandReadAlarm := Ps1AsyncCommandReadAlarmWrapper,
        asyncCommandWriteAlarm := Ps1AsyncCommandWriteAlarmWrapper,
        asyncCommandNullAlarm := Ps1AsyncCommandNullAlarmWrapper,
        setupAlarm := Ps1SetupAlarmWrapper
    );

    Ps1InvalidCommandTypeAlarmWrapper.Setup(REF(Ps1InvalidCommandTypeAlarm));
    Ps1PoppedNullCommandAlarmWrapper.Setup(REF(Ps1PoppedNullCommandAlarm));
    Ps1InvalidCommandAlarmWrapper.Setup(REF(Ps1InvalidCommandAlarm));

    // Setup AsyncInterface with Setup method
    Ps1AsyncInterface.Setup(
        reader := Ps1AsyncReader,
        writer := Ps1AsyncWriter,
        invalidCommandTypeAlarm := Ps1InvalidCommandTypeAlarmWrapper,
        poppedNullCommandAlarm := Ps1PoppedNullCommandAlarmWrapper,
        invalidCommandAlarm := Ps1InvalidCommandAlarmWrapper
    );
    Ps1AsyncInterface.SetListener(PowerSource1);

    Ps1AsyncReaderErrorAlarmWrapper.Setup(REF(Ps1AsyncReaderErrorAlarm));
    Ps1AsyncWriterErrorAlarmWrapper.Setup(REF(Ps1AsyncWriterErrorAlarm));

    Ps1AsyncReader.ErrorAlarm := Ps1AsyncReaderErrorAlarmWrapper;
    Ps1AsyncWriter.ErrorAlarm := Ps1AsyncWriterErrorAlarmWrapper;

    PowerSource1.SetIdentifier(Esab.AssetIdentifier#PowerSource1);
    assetsManager.RegisterAsset(REF(PowerSource1));
END_FUNCTION

PROGRAM PowerSource1IoReadWrite
    VAR_EXTERNAL
        PowerSource1 : Aristo1000.PowerSource;

        PS1_Data : Io;
        I_Pab1 : RawPabToController;
        Q_Pab1 : RawControllerToPab;
        DQ_B_PowerSource1_RemoteStart : BOOL;
    END_VAR

    PabRead(REF(PS1_Data.Pab.Input), REF(I_Pab1));

    PabWrite(REF(PS1_Data.Pab.Output), REF(Q_Pab1));

    PS1_Data.Output.RemoteStart.Write(DQ_B_PowerSource1_RemoteStart);
END_PROGRAM

(* ---- PowerSource2.st ---- *)
USING Esab.WeldSystem.PowerSources;
USING Esab.WeldSystem;
USING Esab.Io;
USING Esab.Utils.Assets;
USING Esab.Utils.Timer;
USING Esab.Utils.Alarming;

USING Siemens.Simatic.S71500.Tasks;
USING Siemens.Simatic.S71500.Alarming;

CONFIGURATION PowerSource2Configuration

    TASK PowerSource2IoTask : ProgramCycle;

    PROGRAM PowerSource2IoProgram WITH PowerSource2IoTask: PowerSource2IoReadWrite;

    // Constants
    VAR_GLOBAL CONSTANT
        PAB2_HWID : WORD := WORD#269;
        PAB2_DEVID : WORD := WORD#264;
    END_VAR

    // Objects
    VAR_GLOBAL
        PowerSource2 : Aristo1000.PowerSource;
        Ps2HeartbeatTimer : OnDelay;
        Ps2Heartbeat : Heartbeat;
        Ps2AsyncInterface : AsyncInterface;
        Ps2AsyncReader : AsyncReader;
        Ps2AsyncWriter : AsyncWriter;
        Ps2AsyncCommands : AsyncCommands;
    END_VAR

    // Alarms
    VAR_GLOBAL
        Ps2ErrorAlarmWrapper : AlarmWrapper;
        {S7.Alarm = NoAck, "Power source 2: Error."}
        Ps2ErrorAlarm : ProgramAlarm;

        Ps2HeartbeatAlarmWrapper : AlarmWrapper;
        {S7.Alarm = NoAck, "Power source 2: No heartbeat."}
        Ps2HeartbeatAlarm : ProgramAlarm;

        Ps2AsyncCommandReadAlarmWrapper : AlarmWrapper;
        {S7.Alarm = NoAck, "Power source 2: Async command (READ) @1%u@ failed."}
        Ps2AsyncCommandReadAlarm : ProgramAlarm;

        Ps2AsyncCommandWriteAlarmWrapper : AlarmWrapper;
        {S7.Alarm = NoAck, "Power source 2: Async command (WRITE) @1%u@ failed."}
        Ps2AsyncCommandWriteAlarm : ProgramAlarm;

        Ps2AsyncCommandNullAlarmWrapper : AlarmWrapper;
        {S7.Alarm = NoAck, "Power source 2: Async command response is NULL."}
        Ps2AsyncCommandNullAlarm : ProgramAlarm;

        Ps2SetupAlarmWrapper : AlarmWrapper;
        {S7.Alarm = NoAck, "Power source 2: Setup error."}
        Ps2SetupAlarm : ProgramAlarm;

        // Ps2 Async Interface Alarms
        Ps2InvalidCommandTypeAlarmWrapper : AlarmWrapper;
        {S7.Alarm = NoAck, "Power source 2 - Async Interface: Invalid command type."}
        Ps2InvalidCommandTypeAlarm : ProgramAlarm;

        Ps2PoppedNullCommandAlarmWrapper : AlarmWrapper;
        {S7.Alarm = NoAck, "Power source 2 - Async Interface: The popped command is NULL."}
        Ps2PoppedNullCommandAlarm : ProgramAlarm;

        Ps2InvalidCommandAlarmWrapper : AlarmWrapper;
        {S7.Alarm = NoAck, "Power source 2 - Async Interface: The type of the popped command is not AsyncCommand."}
        Ps2InvalidCommandAlarm : ProgramAlarm;

        // Ps2 Async Reader Alarms
        Ps2AsyncReaderErrorAlarmWrapper : AlarmWrapper;
        {S7.Alarm = NoAck, "Power source 2 - Async Reader: Error when reading async data, status: @1%u@."}
        Ps2AsyncReaderErrorAlarm : ProgramAlarm;

        // Ps2 Async Writer Alarms
        Ps2AsyncWriterErrorAlarmWrapper : AlarmWrapper;
        {S7.Alarm = NoAck, "Power source 2 - Async Writer: Error when writing async data, status: @1%u@."}
        Ps2AsyncWriterErrorAlarm : ProgramAlarm;
    END_VAR

    // Interface
    VAR_GLOBAL
        {S7.Extern=ReadWrite}
        PS2_Data : Io;
    END_VAR

    // Retained
    VAR_GLOBAL RETAIN
        Ps2RuntimeParameters : RuntimeParameters;
        Ps2HardwareConfiguration : HardwareConfiguration;
    END_VAR
END_CONFIGURATION

FUNCTION InitializePs2
    VAR_INPUT
        assetsManager : IAssetsManager;
    END_VAR

    VAR_EXTERNAL CONSTANT
        PAB2_HWID : WORD;
        PAB2_DEVID : WORD;
    END_VAR

    VAR_EXTERNAL
        PS2_Data : Io;

        PowerSource2 : Aristo1000.PowerSource;
        Ps2HeartbeatTimer : OnDelay;
        Ps2Heartbeat : Heartbeat;
        Ps2AsyncInterface : AsyncInterface;
        Ps2AsyncReader : AsyncReader;
        Ps2AsyncWriter : AsyncWriter;
        Ps2AsyncCommands : AsyncCommands;
        Ps2RuntimeParameters : RuntimeParameters;
        Ps2HardwareConfiguration : HardwareConfiguration;

        Ps2ErrorAlarmWrapper : AlarmWrapper;
        Ps2HeartbeatAlarmWrapper : AlarmWrapper;
        Ps2AsyncCommandReadAlarmWrapper : AlarmWrapper;
        Ps2AsyncCommandWriteAlarmWrapper : AlarmWrapper;
        Ps2AsyncCommandNullAlarmWrapper : AlarmWrapper;
        Ps2SetupAlarmWrapper : AlarmWrapper;

        Ps2ErrorAlarm : ProgramAlarm;
        Ps2HeartbeatAlarm : ProgramAlarm;
        Ps2AsyncCommandReadAlarm : ProgramAlarm;
        Ps2AsyncCommandWriteAlarm : ProgramAlarm;
        Ps2AsyncCommandNullAlarm : ProgramAlarm;
        Ps2SetupAlarm : ProgramAlarm;

        Ps2InvalidCommandTypeAlarmWrapper : AlarmWrapper;
        Ps2PoppedNullCommandAlarmWrapper : AlarmWrapper;
        Ps2InvalidCommandAlarmWrapper : AlarmWrapper;

        Ps2InvalidCommandTypeAlarm : ProgramAlarm;
        Ps2PoppedNullCommandAlarm : ProgramAlarm;
        Ps2InvalidCommandAlarm : ProgramAlarm;

        Ps2AsyncReaderErrorAlarmWrapper : AlarmWrapper;
        Ps2AsyncWriterErrorAlarmWrapper : AlarmWrapper;

        Ps2AsyncReaderErrorAlarm : ProgramAlarm;
        Ps2AsyncWriterErrorAlarm : ProgramAlarm;
    END_VAR

    // Setup heartbeat
    Ps2Heartbeat.Input := PS2_Data.Pab.Input.Heartbeat;
    Ps2Heartbeat.Timer := Ps2HeartbeatTimer;

    // Setup async interface
    Ps2AsyncReader.HwId := PAB2_HWID;
    Ps2AsyncWriter.HwId := PAB2_HWID;

    // Setup alarm wrappers
    Ps2ErrorAlarmWrapper.Setup(REF(Ps2ErrorAlarm));
    Ps2HeartbeatAlarmWrapper.Setup(REF(Ps2HeartbeatAlarm));
    Ps2AsyncCommandReadAlarmWrapper.Setup(REF(Ps2AsyncCommandReadAlarm));
    Ps2AsyncCommandWriteAlarmWrapper.Setup(REF(Ps2AsyncCommandWriteAlarm));
    Ps2AsyncCommandNullAlarmWrapper.Setup(REF(Ps2AsyncCommandNullAlarm));
    Ps2SetupAlarmWrapper.Setup(REF(Ps2SetupAlarm));

    // Setup PowerSource using Setup method
    PowerSource2.Setup(
        id := UINT#2,
        ioDeviceId := PAB2_DEVID,
        heartbeat := Ps2Heartbeat,
        io := REF(PS2_Data),
        runtimeParameters := REF(Ps2RuntimeParameters),
        hardwareConfiguration := REF(Ps2HardwareConfiguration),
        asyncInterface := Ps2AsyncInterface,
        errorAlarm := Ps2ErrorAlarmWrapper,
        heartbeatAlarm := Ps2HeartbeatAlarmWrapper,
        asyncCommandReadAlarm := Ps2AsyncCommandReadAlarmWrapper,
        asyncCommandWriteAlarm := Ps2AsyncCommandWriteAlarmWrapper,
        asyncCommandNullAlarm := Ps2AsyncCommandNullAlarmWrapper,
        setupAlarm := Ps2SetupAlarmWrapper
    );

    Ps2InvalidCommandTypeAlarmWrapper.Setup(REF(Ps2InvalidCommandTypeAlarm));
    Ps2PoppedNullCommandAlarmWrapper.Setup(REF(Ps2PoppedNullCommandAlarm));
    Ps2InvalidCommandAlarmWrapper.Setup(REF(Ps2InvalidCommandAlarm));

    // Setup AsyncInterface with Setup method
    Ps2AsyncInterface.Setup(
        reader := Ps2AsyncReader,
        writer := Ps2AsyncWriter,
        invalidCommandTypeAlarm := Ps2InvalidCommandTypeAlarmWrapper,
        poppedNullCommandAlarm := Ps2PoppedNullCommandAlarmWrapper,
        invalidCommandAlarm := Ps2InvalidCommandAlarmWrapper
    );
    Ps2AsyncInterface.SetListener(PowerSource2);

    Ps2AsyncReaderErrorAlarmWrapper.Setup(REF(Ps2AsyncReaderErrorAlarm));
    Ps2AsyncWriterErrorAlarmWrapper.Setup(REF(Ps2AsyncWriterErrorAlarm));

    Ps2AsyncReader.ErrorAlarm := Ps2AsyncReaderErrorAlarmWrapper;
    Ps2AsyncWriter.ErrorAlarm := Ps2AsyncWriterErrorAlarmWrapper;

    PowerSource2.SetIdentifier(Esab.AssetIdentifier#PowerSource2);
    assetsManager.RegisterAsset(REF(PowerSource2));
END_FUNCTION

PROGRAM PowerSource2IoReadWrite
    VAR_EXTERNAL
        PowerSource2 : Aristo1000.PowerSource;

        PS2_Data : Io;
        I_Pab2 : RawPabToController;
        Q_Pab2 : RawControllerToPab;
        DQ_B_PowerSource2_RemoteStart : BOOL;
    END_VAR

    PabRead(REF(PS2_Data.Pab.Input), REF(I_Pab2));

    PabWrite(REF(PS2_Data.Pab.Output), REF(Q_Pab2));

    PS2_Data.Output.RemoteStart.Write(DQ_B_PowerSource2_RemoteStart);
END_PROGRAM
